KUKA KRL program: EPS_2_251245_SANMH1A_A_20250910012812.src

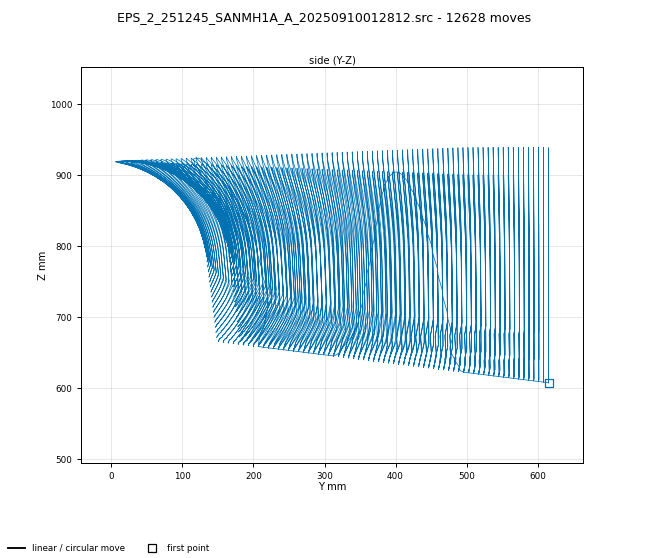
[picture p0: tool path of EPS_2_251245_SANMH1A_A_20250910012812.src, 12628 of 12630 moves have a stored position in this frame; points joined in program order, loops and branches not executed]
&ACCESS RVP
&REL 4
&COMMENT QRS 19112012
&PARAM EDITMASK = *
DEF PART()
EXT BAS (BAS_COMMAND :IN,REAL :IN )
INT I
BAS (#INITMOV,0 )

;KUKA QRS Post kuka4.cps  Date:22-06-2017 !

File_ID=2818

QRS_PRE_INIT()

;Init var - Until changes are made in qrs_pre_init
Outlet_Square_prg=0
Inlet_1_Square_prg=0
Inlet_2_Square_prg=0
Inlet_3_Square_prg=0
Inlet_4_Square_prg=0
Inlet_5_Square_prg=0

Outlet_1={X 0.000, Y 505.360, Z 814.000, B 0.000, E1 0.000 }
Inlet_1={X 0.000, Y 508.180, Z 775.000, B 0.000, E1 175.000 }
Outlet_1_type=251
Inlet_1_type=251
;QRS#1=Sidecore dimensions
;QRS#2=250-10" PVC SDR 35
;QRS#3=250-10" PVC SDR 35
;QRS#4=
;QRS#5=
;QRS#6=
;QRS#7=
;QRS#8=
;QRS#9=14M PSX
;QRS#10=14M PSX
;QRS#11=
;QRS#12=
;QRS#13=
;QRS#14=
;QRS#15=
;QRS#16=1220x127x1219 4'
;QRS#17=EPS Height
;QRS#18=939,5
;QRS#19=*
;QRS#20= UPDATED VERSION 22-06-2017
;QRS#21=*
Outlet_Square=0100
Inlet_1_Square=0100
Inlet_2_Square=0
Inlet_3_Square=0
Inlet_4_Square=0
Inlet_5_Square=0
Mill_Square=1
Outlet_Square_Prg=205
Inlet_1_Square_prg=205

QRS_INIT()

$ADVANCE=5

; T1
PTP {E1 173.423,E2 173.423}
PTP {X 0,Y 615.488,A -85,B 0,C 180,E1 173.423,E2 173.423,E3 0,E4 0,E5 0,E6 0}
QRS_SPEED_INIT()
LIN {X 0,Y 615.488,Z 607.823,A -85,B 0,C 180,E1 173.423,E2 173.423,E3 0,E4 0,E5 0,E6 0} C_VEL
LIN {X 0,Y 615.463,Z 607.814,A -85,B 0,C 180,E1 170.801,E2 170.801} C_VEL
LIN {X 0,Y 615.489,Z 607.808,A -85,B 0,C 180,E1 168.139,E2 168.139} C_VEL
LIN {X 0,Y 615.488,Z 607.825,A -85,B 0,C 180,E1 165.451,E2 165.451} C_VEL
LIN {X 0,Y 615.458,Z 607.816,A -85,B 0,C 180,E1 162.728,E2 162.728} C_VEL
LIN {X 0,Y 615.49,Z 607.808,A -85,B 0,C 180,E1 159.967,E2 159.967} C_VEL
LIN {X 0,Y 615.487,Z 607.825,A -85,B 0,C 180,E1 157.155,E2 157.155} C_VEL
LIN {X 0,Y 615.451,Z 607.816,A -85,B 0,C 180,E1 154.439,E2 154.439} C_VEL
LIN {X 0,Y 615.496,Z 607.811,A -85,B 0,C 180,E1 151.548,E2 151.548} C_VEL
LIN {X 0,Y 615.475,Z 607.824,A -85,B 0,C 180,E1 148.916,E2 148.916} C_VEL
LIN {X 0,Y 615.45,Z 607.819,A -85,B 0,C 180,E1 146.471,E2 146.471} C_VEL
LIN {X 0,Y 615.447,Z 607.816,A -85,B 0,C 180,E1 144.172,E2 144.172} C_VEL
LIN {X 0,Y 615.452,Z 607.814,A -85,B 0,C 180,E1 141.928,E2 141.928} C_VEL
LIN {X 0,Y 615.486,Z 607.812,A -85,B 0,C 180,E1 139.393,E2 139.393} C_VEL
LIN {X 0,Y 615.486,Z 607.824,A -85,B 0,C 180,E1 136.755,E2 136.755} C_VEL
LIN {X 0,Y 615.441,Z 607.819,A -85,B 0,C 180,E1 134.154,E2 134.154} C_VEL
LIN {X 0,Y 615.437,Z 607.819,A -85,B 0,C 180,E1 132.074,E2 132.074} C_VEL
LIN {X 0,Y 615.438,Z 607.817,A -85,B 0,C 180,E1 129.754,E2 129.754} C_VEL
LIN {X 0,Y 615.497,Z 607.816,A -85,B 0,C 180,E1 126.937,E2 126.937} C_VEL
LIN {X 0,Y 615.496,Z 607.823,A -85,B 0,C 180,E1 124.701,E2 124.701} C_VEL
LIN {X 0,Y 615.464,Z 607.823,A -85,B 0,C 180,E1 122.326,E2 122.326} C_VEL
LIN {X 0,Y 615.43,Z 607.82,A -85,B 0,C 180,E1 119.784,E2 119.784} C_VEL
LIN {X 0,Y 615.434,Z 607.822,A -85,B 0,C 180,E1 117.918,E2 117.918} C_VEL
LIN {X 0,Y 615.425,Z 607.82,A -85,B 0,C 180,E1 115.556,E2 115.556} C_VEL
LIN {X 0,Y 615.447,Z 607.824,A -85,B 0,C 180,E1 115.099,E2 115.099} C_VEL
LIN {X 0,Y 615.477,Z 626.453,A -85,B 0,C 180,E1 112.342,E2 112.342} C_VEL
LIN {X 0,Y 615.495,Z 638.775,A -85,B 0,C 180,E1 110.541,E2 110.541} C_VEL
LIN {X 0,Y 615.463,Z 775.158,A -85,B 0,C 180,E1 108.906,E2 108.906} C_VEL
LIN {X 0,Y 615.489,Z 789.394,A -85,B 0,C 180,E1 108.604,E2 108.604} C_VEL
LIN {X 0,Y 615.488,Z 802.541,A -85,B 0,C 180,E1 108.199,E2 108.199} C_VEL
LIN {X 0,Y 615.492,Z 814.87,A -85,B 0,C 180,E1 107.699,E2 107.699} C_VEL
LIN {X 0,Y 615.483,Z 828.082,A -85,B 0,C 180,E1 107.014,E2 107.014} C_VEL
LIN {X 0,Y 615.498,Z 839.221,A -85,B 0,C 180,E1 106.301,E2 106.301} C_VEL
LIN {X 0,Y 615.499,Z 850.82,A -85,B 0,C 180,E1 105.395,E2 105.395} C_VEL
LIN {X 0,Y 615.497,Z 861.349,A -85,B 0,C 180,E1 104.395,E2 104.395} C_VEL
LIN {X 0,Y 615.497,Z 870.257,A -85,B 0,C 180,E1 103.369,E2 103.369} C_VEL
LIN {X 0,Y 615.498,Z 878.577,A -85,B 0,C 180,E1 102.195,E2 102.195} C_VEL
LIN {X 0,Y 615.496,Z 884.373,A -85,B 0,C 180,E1 101.193,E2 101.193} C_VEL
LIN {X 0,Y 615.498,Z 889.088,A -85,B 0,C 180,E1 100.194,E2 100.194} C_VEL
LIN {X 0,Y 615.493,Z 893.953,A -85,B 0,C 180,E1 98.867,E2 98.867} C_VEL
LIN {X 0,Y 615.493,Z 896.596,A -85,B 0,C 180,E1 97.875,E2 97.875} C_VEL
LIN {X 0,Y 615.495,Z 898.88,A -85,B 0,C 180,E1 96.557,E2 96.557} C_VEL
LIN {X 0,Y 615.494,Z 899.826,A -85,B 0,C 180,E1 95.241,E2 95.241} C_VEL
LIN {X 0,Y 615.492,Z 899.459,A -85,B 0,C 180,E1 93.928,E2 93.928} C_VEL
LIN {X 0,Y 615.491,Z 897.783,A -85,B 0,C 180,E1 92.618,E2 92.618} C_VEL
LIN {X 0,Y 615.494,Z 894.753,A -85,B 0,C 180,E1 91.309,E2 91.309} C_VEL
LIN {X 0,Y 615.496,Z 890.297,A -85,B 0,C 180,E1 90,E2 90} C_VEL
LIN {X 0,Y 615.495,Z 885.885,A -85,B 0,C 180,E1 89.019,E2 89.019} C_VEL
LIN {X 0,Y 615.497,Z 880.538,A -85,B 0,C 180,E1 88.037,E2 88.037} C_VEL
LIN {X 0,Y 615.496,Z 872.897,A -85,B 0,C 180,E1 86.891,E2 86.891} C_VEL
LIN {X 0,Y 615.497,Z 863.473,A -85,B 0,C 180,E1 85.744,E2 85.744} C_VEL
LIN {X 0,Y 615.498,Z 853.62,A -85,B 0,C 180,E1 84.759,E2 84.759} C_VEL
LIN {X 0,Y 615.499,Z 842.627,A -85,B 0,C 180,E1 83.855,E2 83.855} C_VEL
LIN {X 0,Y 615.489,Z 830.195,A -85,B 0,C 180,E1 83.022,E2 83.022} C_VEL
LIN {X 0,Y 615.492,Z 818.224,A -85,B 0,C 180,E1 82.372,E2 82.372} C_VEL
LIN {X 0,Y 615.493,Z 804.758,A -85,B 0,C 180,E1 81.794,E2 81.794} C_VEL
LIN {X 0,Y 615.479,Z 790.589,A -85,B 0,C 180,E1 81.339,E2 81.339} C_VEL
LIN {X 0,Y 615.454,Z 776.509,A -85,B 0,C 180,E1 81.028,E2 81.028} C_VEL
LIN {X 0,Y 615.451,Z 738.125,A -85,B 0,C 180,E1 80.552,E2 80.552} C_VEL
LIN {X 0,Y 615.472,Z 638.747,A -85,B 0,C 180,E1 79.364,E2 79.364} C_VEL
LIN {X 0,Y 615.467,Z 620.084,A -85,B 0,C 180,E1 76.63,E2 76.63} C_VEL
LIN {X 0,Y 615.422,Z 607.823,A -85,B 0,C 180,E1 74.793,E2 74.793} C_VEL
LIN {X 0,Y 615.418,Z 607.824,A -85,B 0,C 180,E1 72.727,E2 72.727} C_VEL
LIN {X 0,Y 615.416,Z 607.824,A -85,B 0,C 180,E1 70.66,E2 70.66} C_VEL
LIN {X 0,Y 615.419,Z 607.823,A -85,B 0,C 180,E1 68.565,E2 68.565} C_VEL
LIN {X 0,Y 615.432,Z 607.821,A -85,B 0,C 180,E1 66.005,E2 66.005} C_VEL
LIN {X 0,Y 615.473,Z 607.821,A -85,B 0,C 180,E1 63.555,E2 63.555} C_VEL
LIN {X 0,Y 615.487,Z 607.824,A -85,B 0,C 180,E1 61.342,E2 61.342} C_VEL
LIN {X 0,Y 615.465,Z 607.823,A -85,B 0,C 180,E1 58.918,E2 58.918} C_VEL
LIN {X 0,Y 615.429,Z 607.822,A -85,B 0,C 180,E1 56.475,E2 56.475} C_VEL
LIN {X 0,Y 615.421,Z 607.821,A -85,B 0,C 180,E1 54.176,E2 54.176} C_VEL
LIN {X 0,Y 615.423,Z 607.821,A -85,B 0,C 180,E1 51.927,E2 51.927} C_VEL
LIN {X 0,Y 615.423,Z 607.821,A -85,B 0,C 180,E1 49.919,E2 49.919} C_VEL
LIN {X 0,Y 615.433,Z 607.821,A -85,B 0,C 180,E1 47.642,E2 47.642} C_VEL
LIN {X 0,Y 615.496,Z 607.825,A -85,B 0,C 180,E1 44.932,E2 44.932} C_VEL
LIN {X 0,Y 615.434,Z 607.819,A -85,B 0,C 180,E1 42.074,E2 42.074} C_VEL
LIN {X 0,Y 615.428,Z 607.82,A -85,B 0,C 180,E1 39.755,E2 39.755} C_VEL
LIN {X 0,Y 615.448,Z 607.823,A -85,B 0,C 180,E1 37.245,E2 37.245} C_VEL
LIN {X 0,Y 615.496,Z 607.823,A -85,B 0,C 180,E1 34.701,E2 34.701} C_VEL
LIN {X 0,Y 615.489,Z 607.813,A -85,B 0,C 180,E1 32.331,E2 32.331} C_VEL
LIN {X 0,Y 615.443,Z 607.816,A -85,B 0,C 180,E1 29.787,E2 29.787} C_VEL
LIN {X 0,Y 615.457,Z 607.814,A -85,B 0,C 180,E1 27.917,E2 27.917} C_VEL
LIN {X 0,Y 615.439,Z 607.817,A -85,B 0,C 180,E1 25.559,E2 25.559} C_VEL
LIN {X 0,Y 615.445,Z 607.816,A -85,B 0,C 180,E1 23.558,E2 23.558} C_VEL
LIN {X 0,Y 615.444,Z 607.816,A -85,B 0,C 180,E1 21.434,E2 21.434} C_VEL
LIN {X 0,Y 615.445,Z 607.816,A -85,B 0,C 180,E1 19.34,E2 19.34} C_VEL
LIN {X 0,Y 615.447,Z 607.816,A -85,B 0,C 180,E1 17.272,E2 17.272} C_VEL
LIN {X 0,Y 615.487,Z 607.824,A -85,B 0,C 180,E1 14.549,E2 14.549} C_VEL
LIN {X 0,Y 615.488,Z 607.81,A -85,B 0,C 180,E1 11.861,E2 11.861} C_VEL
LIN {X 0,Y 615.453,Z 607.814,A -85,B 0,C 180,E1 9.2,E2 9.2} C_VEL
LIN {X 0,Y 615.474,Z 607.822,A -85,B 0,C 180,E1 6.557,E2 6.557} C_VEL
LIN {X 0,Y 615.495,Z 607.814,A -85,B 0,C 180,E1 3.929,E2 3.929} C_VEL
LIN {X 0,Y 615.476,Z 607.809,A -85,B 0,C 180,E1 1.309,E2 1.309} C_VEL
LIN {X 0,Y 615.462,Z 607.817,A -85,B 0,C 180,E1 -1.308,E2 -1.308} C_VEL
LIN {X 0,Y 615.492,Z 607.824,A -85,B 0,C 180,E1 -3.928,E2 -3.928} C_VEL
LIN {X 0,Y 615.49,Z 607.808,A -85,B 0,C 180,E1 -6.578,E2 -6.578} C_VEL
LIN {X 0,Y 615.468,Z 607.812,A -85,B 0,C 180,E1 -9.199,E2 -9.199} C_VEL
LIN {X 0,Y 615.486,Z 607.823,A -85,B 0,C 180,E1 -11.861,E2 -11.861} C_VEL
LIN {X 0,Y 615.492,Z 607.81,A -85,B 0,C 180,E1 -14.549,E2 -14.549} C_VEL
LIN {X 0,Y 615.477,Z 607.809,A -85,B 0,C 180,E1 -17.271,E2 -17.271} C_VEL
LIN {X 0,Y 615.491,Z 607.823,A -85,B 0,C 180,E1 -20.033,E2 -20.033} C_VEL
LIN {X 0,Y 615.49,Z 607.808,A -85,B 0,C 180,E1 -22.844,E2 -22.844} C_VEL
LIN {X 0,Y 615.477,Z 607.811,A -85,B 0,C 180,E1 -25.566,E2 -25.566} C_VEL
LIN {X 0,Y 615.496,Z 607.819,A -85,B 0,C 180,E1 -28.451,E2 -28.451} C_VEL
LIN {X 0,Y 615.489,Z 607.807,A -85,B 0,C 180,E1 -31.086,E2 -31.086} C_VEL
LIN {X 0,Y 615.492,Z 607.806,A -85,B 0,C 180,E1 -33.534,E2 -33.534} C_VEL
LIN {X 0,Y 615.49,Z 607.826,A -85,B 0,C 180,E1 -36.425,E2 -36.425} C_VEL
LIN {X 0,Y 615.49,Z 607.809,A -85,B 0,C 180,E1 -39.062,E2 -39.062} C_VEL
LIN {X 0,Y 615.487,Z 607.806,A -85,B 0,C 180,E1 -41.474,E2 -41.474} C_VEL
LIN {X 0,Y 615.484,Z 607.815,A -85,B 0,C 180,E1 -44.15,E2 -44.15} C_VEL
LIN {X 0,Y 615.49,Z 607.814,A -85,B 0,C 180,E1 -46.952,E2 -46.952} C_VEL
LIN {X 0,Y 615.486,Z 607.807,A -85,B 0,C 180,E1 -49.393,E2 -49.393} C_VEL
LIN {X 0,Y 615.487,Z 607.808,A -85,B 0,C 180,E1 -51.988,E2 -51.988} C_VEL
LIN {X 0,Y 615.488,Z 607.816,A -85,B 0,C 180,E1 -54.384,E2 -54.384} C_VEL
LIN {X 0,Y 615.487,Z 607.827,A -85,B 0,C 180,E1 -56.764,E2 -56.764} C_VEL
LIN {X 0,Y 615.484,Z 607.818,A -85,B 0,C 180,E1 -59.08,E2 -59.08} C_VEL
LIN {X 0,Y 615.487,Z 607.808,A -85,B 0,C 180,E1 -61.55,E2 -61.55} C_VEL
LIN {X 0,Y 615.494,Z 607.811,A -85,B 0,C 180,E1 -64.43,E2 -64.43} C_VEL
LIN {X 0,Y 615.488,Z 607.97,A -85,B 0,C 180,E1 -66.162,E2 -66.162} C_VEL
LIN {X 0,Y 615.481,Z 630.471,A -85,B 0,C 180,E1 -68.919,E2 -68.919} C_VEL
LIN {X 0,Y 615.498,Z 653.753,A -85,B 0,C 180,E1 -71.721,E2 -71.721} C_VEL
LIN {X 0,Y 615.495,Z 676.284,A -85,B 0,C 180,E1 -74.392,E2 -74.392} C_VEL
LIN {X 0,Y 615.481,Z 814.24,A -85,B 0,C 180,E1 -76.051,E2 -76.051} C_VEL
LIN {X 0,Y 615.484,Z 827.853,A -85,B 0,C 180,E1 -76.336,E2 -76.336} C_VEL
LIN {X 0,Y 615.491,Z 841.564,A -85,B 0,C 180,E1 -76.757,E2 -76.757} C_VEL
LIN {X 0,Y 615.495,Z 854.834,A -85,B 0,C 180,E1 -77.302,E2 -77.302} C_VEL
LIN {X 0,Y 615.49,Z 867.598,A -85,B 0,C 180,E1 -77.972,E2 -77.972} C_VEL
LIN {X 0,Y 615.499,Z 879.181,A -85,B 0,C 180,E1 -78.724,E2 -78.724} C_VEL
LIN {X 0,Y 615.498,Z 890.747,A -85,B 0,C 180,E1 -79.639,E2 -79.639} C_VEL
LIN {X 0,Y 615.497,Z 901.087,A -85,B 0,C 180,E1 -80.636,E2 -80.636} C_VEL
LIN {X 0,Y 615.497,Z 909.602,A -85,B 0,C 180,E1 -81.629,E2 -81.629} C_VEL
LIN {X 0,Y 615.497,Z 917.726,A -85,B 0,C 180,E1 -82.784,E2 -82.784} C_VEL
LIN {X 0,Y 615.496,Z 923.429,A -85,B 0,C 180,E1 -83.773,E2 -83.773} C_VEL
LIN {X 0,Y 615.495,Z 928.08,A -85,B 0,C 180,E1 -84.759,E2 -84.759} C_VEL
LIN {X 0,Y 615.495,Z 932.901,A -85,B 0,C 180,E1 -86.071,E2 -86.071} C_VEL
LIN {X 0,Y 615.496,Z 936.252,A -85,B 0,C 180,E1 -87.382,E2 -87.382} C_VEL
LIN {X 0,Y 615.489,Z 938.228,A -85,B 0,C 180,E1 -88.691,E2 -88.691} C_VEL
LIN {X 0,Y 615.493,Z 938.889,A -85,B 0,C 180,E1 -90,E2 -90} C_VEL
LIN {X 0,Y 615.489,Z 938.229,A -85,B 0,C 180,E1 -91.309,E2 -91.309} C_VEL
LIN {X 0,Y 615.496,Z 936.252,A -85,B 0,C 180,E1 -92.618,E2 -92.618} C_VEL
LIN {X 0,Y 615.495,Z 932.901,A -85,B 0,C 180,E1 -93.928,E2 -93.928} C_VEL
LIN {X 0,Y 615.495,Z 928.081,A -85,B 0,C 180,E1 -95.241,E2 -95.241} C_VEL
LIN {X 0,Y 615.495,Z 921.628,A -85,B 0,C 180,E1 -96.557,E2 -96.557} C_VEL
LIN {X 0,Y 615.497,Z 914.441,A -85,B 0,C 180,E1 -97.71,E2 -97.71} C_VEL
LIN {X 0,Y 615.497,Z 906.903,A -85,B 0,C 180,E1 -98.702,E2 -98.702} C_VEL
LIN {X 0,Y 615.495,Z 897.853,A -85,B 0,C 180,E1 -99.696,E2 -99.696} C_VEL
LIN {X 0,Y 615.497,Z 887.757,A -85,B 0,C 180,E1 -100.618,E2 -100.618} C_VEL
LIN {X 0,Y 615.498,Z 876.857,A -85,B 0,C 180,E1 -101.443,E2 -101.443} C_VEL
LIN {X 0,Y 615.493,Z 864.705,A -85,B 0,C 180,E1 -102.195,E2 -102.195} C_VEL
LIN {X 0,Y 615.488,Z 851.091,A -85,B 0,C 180,E1 -102.865,E2 -102.865} C_VEL
LIN {X 0,Y 615.489,Z 837.834,A -85,B 0,C 180,E1 -103.369,E2 -103.369} C_VEL
LIN {X 0,Y 615.482,Z 824.286,A -85,B 0,C 180,E1 -103.748,E2 -103.748} C_VEL
LIN {X 0,Y 615.482,Z 810.17,A -85,B 0,C 180,E1 -104.007,E2 -104.007} C_VEL
LIN {X 0,Y 615.495,Z 676.286,A -85,B 0,C 180,E1 -105.608,E2 -105.608} C_VEL
LIN {X 0,Y 615.489,Z 652.401,A -85,B 0,C 180,E1 -108.441,E2 -108.441} C_VEL
LIN {X 0,Y 615.482,Z 629.028,A -85,B 0,C 180,E1 -111.256,E2 -111.256} C_VEL
LIN {X 0,Y 615.487,Z 607.807,A -85,B 0,C 180,E1 -113.866,E2 -113.866} C_VEL
LIN {X 0,Y 615.486,Z 607.808,A -85,B 0,C 180,E1 -116.444,E2 -116.444} C_VEL
LIN {X 0,Y 615.485,Z 607.811,A -85,B 0,C 180,E1 -118.658,E2 -118.658} C_VEL
LIN {X 0,Y 615.488,Z 607.822,A -85,B 0,C 180,E1 -121.086,E2 -121.086} C_VEL
LIN {X 0,Y 615.492,Z 607.807,A -85,B 0,C 180,E1 -124.022,E2 -124.022} C_VEL
LIN {X 0,Y 615.484,Z 607.807,A -85,B 0,C 180,E1 -126.425,E2 -126.425} C_VEL
LIN {X 0,Y 615.481,Z 607.818,A -85,B 0,C 180,E1 -129.061,E2 -129.061} C_VEL
LIN {X 0,Y 615.497,Z 607.824,A -85,B 0,C 180,E1 -131.473,E2 -131.473} C_VEL
LIN {X 0,Y 615.495,Z 607.807,A -85,B 0,C 180,E1 -134.149,E2 -134.149} C_VEL
LIN {X 0,Y 615.492,Z 607.809,A -85,B 0,C 180,E1 -136.952,E2 -136.952} C_VEL
LIN {X 0,Y 615.489,Z 607.82,A -85,B 0,C 180,E1 -139.394,E2 -139.394} C_VEL
LIN {X 0,Y 615.484,Z 607.816,A -85,B 0,C 180,E1 -141.989,E2 -141.989} C_VEL
LIN {X 0,Y 615.491,Z 607.807,A -85,B 0,C 180,E1 -144.384,E2 -144.384} C_VEL
LIN {X 0,Y 615.491,Z 607.805,A -85,B 0,C 180,E1 -146.764,E2 -146.764} C_VEL
LIN {X 0,Y 615.49,Z 607.808,A -85,B 0,C 180,E1 -149.08,E2 -149.08} C_VEL
LIN {X 0,Y 615.494,Z 607.817,A -85,B 0,C 180,E1 -151.549,E2 -151.549} C_VEL
LIN {X 0,Y 615.48,Z 607.812,A -85,B 0,C 180,E1 -154.433,E2 -154.433} C_VEL
LIN {X 0,Y 615.49,Z 607.807,A -85,B 0,C 180,E1 -157.156,E2 -157.156} C_VEL
LIN {X 0,Y 615.49,Z 607.827,A -85,B 0,C 180,E1 -159.967,E2 -159.967} C_VEL
LIN {X 0,Y 615.48,Z 607.81,A -85,B 0,C 180,E1 -162.729,E2 -162.729} C_VEL
LIN {X 0,Y 615.492,Z 607.808,A -85,B 0,C 180,E1 -165.451,E2 -165.451} C_VEL
LIN {X 0,Y 615.489,Z 607.827,A -85,B 0,C 180,E1 -168.139,E2 -168.139} C_VEL
LIN {X 0,Y 615.473,Z 607.812,A -85,B 0,C 180,E1 -170.801,E2 -170.801} C_VEL
LIN {X 0,Y 615.491,Z 607.806,A -85,B 0,C 180,E1 -173.444,E2 -173.444} C_VEL
LIN {X 0,Y 615.495,Z 607.819,A -85,B 0,C 180,E1 -176.072,E2 -176.072} C_VEL
LIN {X 0,Y 615.472,Z 607.818,A -85,B 0,C 180,E1 -178.692,E2 -178.692} C_VEL
LIN {X 0,Y 615.479,Z 607.808,A -85,B 0,C 180,E1 -181.309,E2 -181.309} C_VEL
LIN {X 0,Y 615.495,Z 607.81,A -85,B 0,C 180,E1 -183.929,E2 -183.929} C_VEL
LIN {X 0,Y 615.488,Z 607.823,A -85,B 0,C 180,E1 -186.577,E2 -186.577} C_VEL
LIN {X 0,Y 614.795,Z 607.961,A -85,B 0,C 180,E1 -187.123,E2 -187.123} C_VEL
LIN {X 0,Y 611.945,Z 608.38,A -85,B 0,C 180,E1 -188.009,E2 -188.009} C_VEL
LIN {X 0,Y 609.556,Z 608.688,A -85,B 0,C 180,E1 -188.722,E2 -188.722} C_VEL
LIN {X 0,Y 608.532,Z 608.803,A -85,B 0,C 180,E1 -189.271,E2 -189.271} C_VEL
LIN {X 0,Y 608.449,Z 608.812,A -85,B 0,C 180,E1 -189.457,E2 -189.457} C_VEL
LIN {X 0,Y 608.466,Z 608.812,A -85,B 0,C 180,E1 -192,E2 -192} C_VEL
LIN {X 0,Y 608.47,Z 608.819,A -85,B 0,C 180,E1 -194.721,E2 -194.721} C_VEL
LIN {X 0,Y 608.437,Z 608.814,A -85,B 0,C 180,E1 -197.477,E2 -197.477} C_VEL
LIN {X 0,Y 608.436,Z 608.814,A -85,B 0,C 180,E1 -199.571,E2 -199.571} C_VEL
LIN {X 0,Y 608.48,Z 608.813,A -85,B 0,C 180,E1 -202.405,E2 -202.405} C_VEL
LIN {X 0,Y 608.455,Z 608.818,A -85,B 0,C 180,E1 -204.571,E2 -204.571} C_VEL
LIN {X 0,Y 608.433,Z 608.815,A -85,B 0,C 180,E1 -207.519,E2 -207.519} C_VEL
LIN {X 0,Y 608.445,Z 608.812,A -85,B 0,C 180,E1 -209.968,E2 -209.968} C_VEL
LIN {X 0,Y 608.454,Z 608.822,A -85,B 0,C 180,E1 -212.88,E2 -212.88} C_VEL
LIN {X 0,Y 608.426,Z 608.821,A -85,B 0,C 180,E1 -215.279,E2 -215.279} C_VEL
LIN {X 0,Y 608.443,Z 608.814,A -85,B 0,C 180,E1 -217.749,E2 -217.749} C_VEL
LIN {X 0,Y 608.435,Z 608.814,A -85,B 0,C 180,E1 -220.327,E2 -220.327} C_VEL
LIN {X 0,Y 608.472,Z 608.817,A -85,B 0,C 180,E1 -223.309,E2 -223.309} C_VEL
LIN {X 0,Y 608.435,Z 608.814,A -85,B 0,C 180,E1 -226.127,E2 -226.127} C_VEL
LIN {X 0,Y 608.452,Z 608.816,A -85,B 0,C 180,E1 -228.823,E2 -228.823} C_VEL
LIN {X 0,Y 608.436,Z 608.817,A -85,B 0,C 180,E1 -231.764,E2 -231.764} C_VEL
LIN {X 0,Y 608.431,Z 608.816,A -85,B 0,C 180,E1 -233.957,E2 -233.957} C_VEL
LIN {X 0,Y 608.413,Z 608.816,A -85,B 0,C 180,E1 -236.326,E2 -236.326} C_VEL
LIN {X 0,Y 608.439,Z 608.814,A -85,B 0,C 180,E1 -238.734,E2 -238.734} C_VEL
LIN {X 0,Y 608.434,Z 608.821,A -85,B 0,C 180,E1 -241.732,E2 -241.732} C_VEL
LIN {X 0,Y 608.424,Z 608.817,A -85,B 0,C 180,E1 -244.289,E2 -244.289} C_VEL
LIN {X 0,Y 608.453,Z 609.014,A -85,B 0,C 180,E1 -244.836,E2 -244.836} C_VEL
LIN {X 0,Y 608.511,Z 625.068,A -85,B 0,C 180,E1 -247.238,E2 -247.238} C_VEL
LIN {X 0,Y 608.498,Z 638.922,A -85,B 0,C 180,E1 -249.283,E2 -249.283} C_VEL
LIN {X 0,Y 608.588,Z 756.65,A -85,B 0,C 180,E1 -250.697,E2 -250.697} C_VEL
LIN {X 0,Y 608.588,Z 777.773,A -85,B 0,C 180,E1 -250.982,E2 -250.982} C_VEL
LIN {X 0,Y 608.58,Z 792.407,A -85,B 0,C 180,E1 -251.323,E2 -251.323} C_VEL
LIN {X 0,Y 608.575,Z 806.351,A -85,B 0,C 180,E1 -251.791,E2 -251.791} C_VEL
LIN {X 0,Y 608.543,Z 819.031,A -85,B 0,C 180,E1 -252.353,E2 -252.353} C_VEL
LIN {X 0,Y 608.527,Z 831.481,A -85,B 0,C 180,E1 -253.045,E2 -253.045} C_VEL
LIN {X 0,Y 608.509,Z 842.188,A -85,B 0,C 180,E1 -253.774,E2 -253.774} C_VEL
LIN {X 0,Y 608.491,Z 852.284,A -85,B 0,C 180,E1 -254.595,E2 -254.595} C_VEL
LIN {X 0,Y 608.475,Z 862.8,A -85,B 0,C 180,E1 -255.621,E2 -255.621} C_VEL
LIN {X 0,Y 608.462,Z 871.428,A -85,B 0,C 180,E1 -256.644,E2 -256.644} C_VEL
LIN {X 0,Y 608.441,Z 879.631,A -85,B 0,C 180,E1 -257.831,E2 -257.831} C_VEL
LIN {X 0,Y 608.432,Z 886.464,A -85,B 0,C 180,E1 -259.065,E2 -259.065} C_VEL
LIN {X 0,Y 608.428,Z 892.015,A -85,B 0,C 180,E1 -260.358,E2 -260.358} C_VEL
LIN {X 0,Y 608.426,Z 895.325,A -85,B 0,C 180,E1 -261.364,E2 -261.364} C_VEL
LIN {X 0,Y 608.421,Z 898.403,A -85,B 0,C 180,E1 -262.7,E2 -262.7} C_VEL
LIN {X 0,Y 608.432,Z 900.085,A -85,B 0,C 180,E1 -264.033,E2 -264.033} C_VEL
LIN {X 0,Y 608.424,Z 900.432,A -85,B 0,C 180,E1 -265.362,E2 -265.362} C_VEL
LIN {X 0,Y 608.416,Z 899.453,A -85,B 0,C 180,E1 -266.689,E2 -266.689} C_VEL
LIN {X 0,Y 608.443,Z 897.137,A -85,B 0,C 180,E1 -268.014,E2 -268.014} C_VEL
LIN {X 0,Y 608.437,Z 893.423,A -85,B 0,C 180,E1 -269.338,E2 -269.338} C_VEL
LIN {X 0,Y 608.437,Z 888.216,A -85,B 0,C 180,E1 -270.662,E2 -270.662} C_VEL
LIN {X 0,Y 608.441,Z 883.177,A -85,B 0,C 180,E1 -271.655,E2 -271.655} C_VEL
LIN {X 0,Y 608.446,Z 876.008,A -85,B 0,C 180,E1 -272.814,E2 -272.814} C_VEL
LIN {X 0,Y 608.455,Z 867.176,A -85,B 0,C 180,E1 -273.974,E2 -273.974} C_VEL
LIN {X 0,Y 608.474,Z 857.942,A -85,B 0,C 180,E1 -274.97,E2 -274.97} C_VEL
LIN {X 0,Y 608.497,Z 846.693,A -85,B 0,C 180,E1 -275.967,E2 -275.967} C_VEL
LIN {X 0,Y 608.535,Z 834.522,A -85,B 0,C 180,E1 -276.849,E2 -276.849} C_VEL
LIN {X 0,Y 608.541,Z 822.682,A -85,B 0,C 180,E1 -277.549,E2 -277.549} C_VEL
LIN {X 0,Y 608.572,Z 810.417,A -85,B 0,C 180,E1 -278.133,E2 -278.133} C_VEL
LIN {X 0,Y 608.585,Z 796.855,A -85,B 0,C 180,E1 -278.634,E2 -278.634} C_VEL
LIN {X 0,Y 608.566,Z 782.762,A -85,B 0,C 180,E1 -279.011,E2 -279.011} C_VEL
LIN {X 0,Y 608.57,Z 769.26,A -85,B 0,C 180,E1 -279.242,E2 -279.242} C_VEL
LIN {X 0,Y 608.587,Z 639.744,A -85,B 0,C 180,E1 -280.792,E2 -280.792} C_VEL
LIN {X 0,Y 608.477,Z 638.817,A -85,B 0,C 180,E1 -280.823,E2 -280.823} C_VEL
LIN {X 0,Y 608.487,Z 621.681,A -85,B 0,C 180,E1 -283.356,E2 -283.356} C_VEL
LIN {X 0,Y 608.423,Z 608.855,A -85,B 0,C 180,E1 -285.279,E2 -285.279} C_VEL
LIN {X 0,Y 608.398,Z 608.819,A -85,B 0,C 180,E1 -287.478,E2 -287.478} C_VEL
LIN {X 0,Y 608.397,Z 608.819,A -85,B 0,C 180,E1 -289.573,E2 -289.573} C_VEL
LIN {X 0,Y 608.418,Z 608.816,A -85,B 0,C 180,E1 -291.694,E2 -291.694} C_VEL
LIN {X 0,Y 608.431,Z 608.823,A -85,B 0,C 180,E1 -294.572,E2 -294.572} C_VEL
LIN {X 0,Y 608.405,Z 608.818,A -85,B 0,C 180,E1 -297.52,E2 -297.52} C_VEL
LIN {X 0,Y 608.407,Z 608.817,A -85,B 0,C 180,E1 -299.783,E2 -299.783} C_VEL
LIN {X 0,Y 608.441,Z 608.819,A -85,B 0,C 180,E1 -302.518,E2 -302.518} C_VEL
LIN {X 0,Y 608.417,Z 608.82,A -85,B 0,C 180,E1 -305.28,E2 -305.28} C_VEL
LIN {X 0,Y 608.404,Z 608.818,A -85,B 0,C 180,E1 -307.751,E2 -307.751} C_VEL
LIN {X 0,Y 608.405,Z 608.819,A -85,B 0,C 180,E1 -310.323,E2 -310.323} C_VEL
LIN {X 0,Y 608.453,Z 608.822,A -85,B 0,C 180,E1 -312.96,E2 -312.96} C_VEL
LIN {X 0,Y 608.415,Z 608.817,A -85,B 0,C 180,E1 -315.74,E2 -315.74} C_VEL
LIN {X 0,Y 608.418,Z 608.816,A -85,B 0,C 180,E1 -317.935,E2 -317.935} C_VEL
LIN {X 0,Y 608.424,Z 608.819,A -85,B 0,C 180,E1 -320.708,E2 -320.708} C_VEL
LIN {X 0,Y 608.445,Z 608.822,A -85,B 0,C 180,E1 -323.084,E2 -323.084} C_VEL
LIN {X 0,Y 608.466,Z 608.816,A -85,B 0,C 180,E1 -325.53,E2 -325.53} C_VEL
LIN {X 0,Y 608.453,Z 608.813,A -85,B 0,C 180,E1 -327.904,E2 -327.904} C_VEL
LIN {X 0,Y 608.431,Z 608.814,A -85,B 0,C 180,E1 -330.218,E2 -330.218} C_VEL
LIN {X 0,Y 608.422,Z 608.816,A -85,B 0,C 180,E1 -332.48,E2 -332.48} C_VEL
LIN {X 0,Y 608.447,Z 608.823,A -85,B 0,C 180,E1 -335.428,E2 -335.428} C_VEL
LIN {X 0,Y 608.449,Z 608.812,A -85,B 0,C 180,E1 -338.307,E2 -338.307} C_VEL
LIN {X 0,Y 608.428,Z 608.815,A -85,B 0,C 180,E1 -340.428,E2 -340.428} C_VEL
LIN {X 0,Y 608.43,Z 608.814,A -85,B 0,C 180,E1 -342.522,E2 -342.522} C_VEL
LIN {X 0,Y 608.468,Z 608.816,A -85,B 0,C 180,E1 -345.279,E2 -345.279} C_VEL
LIN {X 0,Y 608.463,Z 608.814,A -85,B 0,C 180,E1 -348,E2 -348} C_VEL
LIN {X 0,Y 608.447,Z 608.812,A -85,B 0,C 180,E1 -350.694,E2 -350.694} C_VEL
LIN {X 0,Y 608.433,Z 608.814,A -85,B 0,C 180,E1 -352.7,E2 -352.7} C_VEL
LIN {X 0,Y 608.437,Z 608.818,A -85,B 0,C 180,E1 -355.362,E2 -355.362} C_VEL
LIN {X 0,Y 608.466,Z 608.817,A -85,B 0,C 180,E1 -358.014,E2 -358.014} C_VEL
LIN {X 0,Y 608.476,Z 608.809,A -85,B 0,C 180,E1 -360.662,E2 -360.662} C_VEL
LIN {X 0,Y 608.458,Z 608.813,A -85,B 0,C 180,E1 -363.311,E2 -363.311} C_VEL
LIN {X 0,Y 608.472,Z 608.819,A -85,B 0,C 180,E1 -365.967,E2 -365.967} C_VEL
LIN {X 0,Y 608.46,Z 608.812,A -85,B 0,C 180,E1 -368.636,E2 -368.636} C_VEL
LIN {X 0,Y 608.437,Z 608.815,A -85,B 0,C 180,E1 -371.324,E2 -371.324} C_VEL
LIN {X 0,Y 608.473,Z 608.821,A -85,B 0,C 180,E1 -374.037,E2 -374.037} C_VEL
LIN {X 0,Y 608.476,Z 608.81,A -85,B 0,C 180,E1 -376.783,E2 -376.783} C_VEL
LIN {X 0,Y 608.449,Z 608.814,A -85,B 0,C 180,E1 -379.571,E2 -379.571} C_VEL
LIN {X 0,Y 608.48,Z 608.815,A -85,B 0,C 180,E1 -382.405,E2 -382.405} C_VEL
LIN {X 0,Y 608.459,Z 608.816,A -85,B 0,C 180,E1 -384.571,E2 -384.571} C_VEL
LIN {X 0,Y 608.482,Z 608.808,A -85,B 0,C 180,E1 -387.207,E2 -387.207} C_VEL
LIN {X 0,Y 608.462,Z 608.816,A -85,B 0,C 180,E1 -389.97,E2 -389.97} C_VEL
LIN {X 0,Y 608.463,Z 608.813,A -85,B 0,C 180,E1 -392.879,E2 -392.879} C_VEL
LIN {X 0,Y 608.451,Z 608.812,A -85,B 0,C 180,E1 -395.277,E2 -395.277} C_VEL
LIN {X 0,Y 608.468,Z 608.811,A -85,B 0,C 180,E1 -397.746,E2 -397.746} C_VEL
LIN {X 0,Y 608.452,Z 608.82,A -85,B 0,C 180,E1 -400.329,E2 -400.329} C_VEL
LIN {X 0,Y 608.474,Z 608.809,A -85,B 0,C 180,E1 -403.309,E2 -403.309} C_VEL
LIN {X 0,Y 608.472,Z 608.813,A -85,B 0,C 180,E1 -406.131,E2 -406.131} C_VEL
LIN {X 0,Y 608.463,Z 608.818,A -85,B 0,C 180,E1 -408.824,E2 -408.824} C_VEL
LIN {X 0,Y 608.47,Z 608.81,A -85,B 0,C 180,E1 -411.759,E2 -411.759} C_VEL
LIN {X 0,Y 608.48,Z 608.809,A -85,B 0,C 180,E1 -413.95,E2 -413.95} C_VEL
LIN {X 0,Y 608.467,Z 608.814,A -85,B 0,C 180,E1 -416.329,E2 -416.329} C_VEL
LIN {X 0,Y 608.48,Z 608.819,A -85,B 0,C 180,E1 -418.727,E2 -418.727} C_VEL
LIN {X 0,Y 608.473,Z 608.811,A -85,B 0,C 180,E1 -421.38,E2 -421.38} C_VEL
LIN {X 0,Y 608.481,Z 608.81,A -85,B 0,C 180,E1 -424.277,E2 -424.277} C_VEL
LIN {X 0,Y 608.475,Z 608.889,A -85,B 0,C 180,E1 -425.985,E2 -425.985} C_VEL
LIN {X 0,Y 608.599,Z 621.803,A -85,B 0,C 180,E1 -427.599,E2 -427.599} C_VEL
LIN {X 0,Y 608.576,Z 644.918,A -85,B 0,C 180,E1 -430.433,E2 -430.433} C_VEL
LIN {X 0,Y 608.521,Z 668.034,A -85,B 0,C 180,E1 -433.218,E2 -433.218} C_VEL
LIN {X 0,Y 608.537,Z 676.431,A -85,B 0,C 180,E1 -434.22,E2 -434.22} C_VEL
LIN {X 0,Y 608.601,Z 814.446,A -85,B 0,C 180,E1 -435.894,E2 -435.894} C_VEL
LIN {X 0,Y 608.581,Z 828.62,A -85,B 0,C 180,E1 -436.199,E2 -436.199} C_VEL
LIN {X 0,Y 608.578,Z 842.707,A -85,B 0,C 180,E1 -436.646,E2 -436.646} C_VEL
LIN {X 0,Y 608.556,Z 854.88,A -85,B 0,C 180,E1 -437.155,E2 -437.155} C_VEL
LIN {X 0,Y 608.519,Z 867.678,A -85,B 0,C 180,E1 -437.832,E2 -437.832} C_VEL
LIN {X 0,Y 608.499,Z 880.469,A -85,B 0,C 180,E1 -438.677,E2 -438.677} C_VEL
LIN {X 0,Y 608.496,Z 890.929,A -85,B 0,C 180,E1 -439.519,E2 -439.519} C_VEL
LIN {X 0,Y 608.479,Z 901.333,A -85,B 0,C 180,E1 -440.527,E2 -440.527} C_VEL
LIN {X 0,Y 608.464,Z 909.913,A -85,B 0,C 180,E1 -441.531,E2 -441.531} C_VEL
LIN {X 0,Y 608.461,Z 918.113,A -85,B 0,C 180,E1 -442.7,E2 -442.7} C_VEL
LIN {X 0,Y 608.443,Z 924.545,A -85,B 0,C 180,E1 -443.831,E2 -443.831} C_VEL
LIN {X 0,Y 608.435,Z 929.961,A -85,B 0,C 180,E1 -445.03,E2 -445.03} C_VEL
LIN {X 0,Y 608.433,Z 933.441,A -85,B 0,C 180,E1 -446.026,E2 -446.026} C_VEL
LIN {X 0,Y 608.424,Z 936.831,A -85,B 0,C 180,E1 -447.352,E2 -447.352} C_VEL
LIN {X 0,Y 608.442,Z 938.83,A -85,B 0,C 180,E1 -448.676,E2 -448.676} C_VEL
LIN {X 0,Y 608.433,Z 939.5,A -85,B 0,C 180,E1 -450,E2 -450} C_VEL
LIN {X 0,Y 608.442,Z 938.83,A -85,B 0,C 180,E1 -451.324,E2 -451.324} C_VEL
LIN {X 0,Y 608.424,Z 936.831,A -85,B 0,C 180,E1 -452.648,E2 -452.648} C_VEL
LIN {X 0,Y 608.433,Z 933.441,A -85,B 0,C 180,E1 -453.974,E2 -453.974} C_VEL
LIN {X 0,Y 608.439,Z 928.568,A -85,B 0,C 180,E1 -455.302,E2 -455.302} C_VEL
LIN {X 0,Y 608.445,Z 922.211,A -85,B 0,C 180,E1 -456.603,E2 -456.603} C_VEL
LIN {X 0,Y 608.453,Z 914.798,A -85,B 0,C 180,E1 -457.8,E2 -457.8} C_VEL
LIN {X 0,Y 608.473,Z 905.823,A -85,B 0,C 180,E1 -458.971,E2 -458.971} C_VEL
LIN {X 0,Y 608.472,Z 896.391,A -85,B 0,C 180,E1 -459.977,E2 -459.977} C_VEL
LIN {X 0,Y 608.506,Z 885.047,A -85,B 0,C 180,E1 -460.973,E2 -460.973} C_VEL
LIN {X 0,Y 608.531,Z 873.147,A -85,B 0,C 180,E1 -461.829,E2 -461.829} C_VEL
LIN {X 0,Y 608.535,Z 860.072,A -85,B 0,C 180,E1 -462.591,E2 -462.591} C_VEL
LIN {X 0,Y 608.557,Z 847.172,A -85,B 0,C 180,E1 -463.184,E2 -463.184} C_VEL
LIN {X 0,Y 608.584,Z 833.18,A -85,B 0,C 180,E1 -463.673,E2 -463.673} C_VEL
LIN {X 0,Y 608.598,Z 819.451,A -85,B 0,C 180,E1 -464.013,E2 -464.013} C_VEL
LIN {X 0,Y 608.622,Z 803.162,A -85,B 0,C 180,E1 -464.257,E2 -464.257} C_VEL
LIN {X 0,Y 608.529,Z 676.432,A -85,B 0,C 180,E1 -465.78,E2 -465.78} C_VEL
LIN {X 0,Y 608.551,Z 653.767,A -85,B 0,C 180,E1 -468.496,E2 -468.496} C_VEL
LIN {X 0,Y 608.573,Z 630.473,A -85,B 0,C 180,E1 -471.332,E2 -471.332} C_VEL
LIN {X 0,Y 608.642,Z 610.247,A -85,B 0,C 180,E1 -473.838,E2 -473.838} C_VEL
LIN {X 0,Y 608.477,Z 608.811,A -85,B 0,C 180,E1 -474.043,E2 -474.043} C_VEL
LIN {X 0,Y 608.449,Z 608.817,A -85,B 0,C 180,E1 -476.774,E2 -476.774} C_VEL
LIN {X 0,Y 608.472,Z 608.817,A -85,B 0,C 180,E1 -479.02,E2 -479.02} C_VEL
LIN {X 0,Y 608.479,Z 608.819,A -85,B 0,C 180,E1 -481.316,E2 -481.316} C_VEL
LIN {X 0,Y 608.477,Z 608.812,A -85,B 0,C 180,E1 -483.735,E2 -483.735} C_VEL
LIN {X 0,Y 608.479,Z 608.809,A -85,B 0,C 180,E1 -486.09,E2 -486.09} C_VEL
LIN {X 0,Y 608.472,Z 608.81,A -85,B 0,C 180,E1 -488.588,E2 -488.588} C_VEL
LIN {X 0,Y 608.47,Z 608.819,A -85,B 0,C 180,E1 -491.343,E2 -491.343} C_VEL
LIN {X 0,Y 608.464,Z 608.811,A -85,B 0,C 180,E1 -494.265,E2 -494.265} C_VEL
LIN {X 0,Y 608.459,Z 608.814,A -85,B 0,C 180,E1 -497.041,E2 -497.041} C_VEL
LIN {X 0,Y 608.453,Z 608.821,A -85,B 0,C 180,E1 -499.697,E2 -499.697} C_VEL
LIN {X 0,Y 608.469,Z 608.811,A -85,B 0,C 180,E1 -502.254,E2 -502.254} C_VEL
LIN {X 0,Y 608.487,Z 608.809,A -85,B 0,C 180,E1 -505.09,E2 -505.09} C_VEL
LIN {X 0,Y 608.473,Z 608.817,A -85,B 0,C 180,E1 -507.906,E2 -507.906} C_VEL
LIN {X 0,Y 608.466,Z 608.814,A -85,B 0,C 180,E1 -510.22,E2 -510.22} C_VEL
LIN {X 0,Y 608.482,Z 608.808,A -85,B 0,C 180,E1 -512.792,E2 -512.792} C_VEL
LIN {X 0,Y 608.485,Z 608.819,A -85,B 0,C 180,E1 -515.846,E2 -515.846} C_VEL
LIN {X 0,Y 608.469,Z 608.814,A -85,B 0,C 180,E1 -518.309,E2 -518.309} C_VEL
LIN {X 0,Y 608.458,Z 608.811,A -85,B 0,C 180,E1 -521.131,E2 -521.131} C_VEL
LIN {X 0,Y 608.466,Z 608.819,A -85,B 0,C 180,E1 -523.906,E2 -523.906} C_VEL
LIN {X 0,Y 608.458,Z 608.813,A -85,B 0,C 180,E1 -526.644,E2 -526.644} C_VEL
LIN {X 0,Y 608.467,Z 608.81,A -85,B 0,C 180,E1 -529.35,E2 -529.35} C_VEL
LIN {X 0,Y 608.478,Z 608.817,A -85,B 0,C 180,E1 -532.033,E2 -532.033} C_VEL
LIN {X 0,Y 608.452,Z 608.815,A -85,B 0,C 180,E1 -534.698,E2 -534.698} C_VEL
LIN {X 0,Y 608.483,Z 608.808,A -85,B 0,C 180,E1 -537.352,E2 -537.352} C_VEL
LIN {X 0,Y 608.478,Z 608.814,A -85,B 0,C 180,E1 -540,E2 -540} C_VEL
LIN {X 0,Y 608.47,Z 608.816,A -85,B 0,C 180,E1 -542.648,E2 -542.648} C_VEL
LIN {X 0,Y 608.451,Z 608.812,A -85,B 0,C 180,E1 -545.302,E2 -545.302} C_VEL
LIN {X 0,Y 608.485,Z 608.81,A -85,B 0,C 180,E1 -547.967,E2 -547.967} C_VEL
LIN {X 0,Y 608.449,Z 608.812,A -85,B 0,C 180,E1 -549.457,E2 -549.457} C_VEL
LIN {X 0,Y 607.785,Z 608.899,A -85,B 0,C 180,E1 -550.01,E2 -550.01} C_VEL
LIN {X 0,Y 604.939,Z 609.254,A -85,B 0,C 180,E1 -550.907,E2 -550.907} C_VEL
LIN {X 0,Y 602.532,Z 609.553,A -85,B 0,C 180,E1 -551.628,E2 -551.628} C_VEL
LIN {X 0,Y 601.496,Z 609.683,A -85,B 0,C 180,E1 -552.185,E2 -552.185} C_VEL
LIN {X 0,Y 601.41,Z 609.692,A -85,B 0,C 180,E1 -552.373,E2 -552.373} C_VEL
LIN {X 0,Y 601.423,Z 609.693,A -85,B 0,C 180,E1 -554.897,E2 -554.897} C_VEL
LIN {X 0,Y 601.429,Z 609.692,A -85,B 0,C 180,E1 -556.986,E2 -556.986} C_VEL
LIN {X 0,Y 601.399,Z 609.69,A -85,B 0,C 180,E1 -559.81,E2 -559.81} C_VEL
LIN {X 0,Y 601.418,Z 609.696,A -85,B 0,C 180,E1 -562.606,E2 -562.606} C_VEL
LIN {X 0,Y 601.394,Z 609.701,A -85,B 0,C 180,E1 -564.879,E2 -564.879} C_VEL
LIN {X 0,Y 601.391,Z 609.694,A -85,B 0,C 180,E1 -567.358,E2 -567.358} C_VEL
LIN {X 0,Y 601.401,Z 609.692,A -85,B 0,C 180,E1 -569.394,E2 -569.394} C_VEL
LIN {X 0,Y 601.396,Z 609.691,A -85,B 0,C 180,E1 -571.728,E2 -571.728} C_VEL
LIN {X 0,Y 601.413,Z 609.689,A -85,B 0,C 180,E1 -574.12,E2 -574.12} C_VEL
LIN {X 0,Y 601.435,Z 609.691,A -85,B 0,C 180,E1 -577.382,E2 -577.382} C_VEL
LIN {X 0,Y 601.4,Z 609.69,A -85,B 0,C 180,E1 -579.996,E2 -579.996} C_VEL
LIN {X 0,Y 601.39,Z 609.695,A -85,B 0,C 180,E1 -582.673,E2 -582.673} C_VEL
LIN {X 0,Y 601.402,Z 609.696,A -85,B 0,C 180,E1 -585.48,E2 -585.48} C_VEL
LIN {X 0,Y 601.409,Z 609.69,A -85,B 0,C 180,E1 -588.409,E2 -588.409} C_VEL
LIN {X 0,Y 601.402,Z 609.697,A -85,B 0,C 180,E1 -591.533,E2 -591.533} C_VEL
LIN {X 0,Y 601.392,Z 609.695,A -85,B 0,C 180,E1 -593.741,E2 -593.741} C_VEL
LIN {X 0,Y 601.406,Z 609.691,A -85,B 0,C 180,E1 -596.069,E2 -596.069} C_VEL
LIN {X 0,Y 601.39,Z 609.692,A -85,B 0,C 180,E1 -598.551,E2 -598.551} C_VEL
LIN {X 0,Y 601.434,Z 609.696,A -85,B 0,C 180,E1 -601.373,E2 -601.373} C_VEL
LIN {X 0,Y 601.375,Z 609.695,A -85,B 0,C 180,E1 -604.38,E2 -604.38} C_VEL
LIN {X 0,Y 601.387,Z 609.778,A -85,B 0,C 180,E1 -604.705,E2 -604.705} C_VEL
LIN {X 0,Y 601.509,Z 619.788,A -85,B 0,C 180,E1 -606.228,E2 -606.228} C_VEL
LIN {X 0,Y 601.509,Z 638.445,A -85,B 0,C 180,E1 -609.024,E2 -609.024} C_VEL
LIN {X 0,Y 601.495,Z 638.915,A -85,B 0,C 180,E1 -609.094,E2 -609.094} C_VEL
LIN {X 0,Y 601.838,Z 644.286,A -85,B 0,C 180,E1 -609.172,E2 -609.172} C_VEL
LIN {X 0,Y 601.719,Z 775.68,A -85,B 0,C 180,E1 -610.778,E2 -610.778} C_VEL
LIN {X 0,Y 601.704,Z 789.973,A -85,B 0,C 180,E1 -611.094,E2 -611.094} C_VEL
LIN {X 0,Y 601.652,Z 802.874,A -85,B 0,C 180,E1 -611.502,E2 -611.502} C_VEL
LIN {X 0,Y 601.591,Z 815.987,A -85,B 0,C 180,E1 -612.054,E2 -612.054} C_VEL
LIN {X 0,Y 601.551,Z 829.026,A -85,B 0,C 180,E1 -612.755,E2 -612.755} C_VEL
LIN {X 0,Y 601.5,Z 841.505,A -85,B 0,C 180,E1 -613.591,E2 -613.591} C_VEL
LIN {X 0,Y 601.485,Z 851.592,A -85,B 0,C 180,E1 -614.411,E2 -614.411} C_VEL
LIN {X 0,Y 601.443,Z 862.236,A -85,B 0,C 180,E1 -615.45,E2 -615.45} C_VEL
LIN {X 0,Y 601.4,Z 870.973,A -85,B 0,C 180,E1 -616.484,E2 -616.484} C_VEL
LIN {X 0,Y 601.381,Z 879.272,A -85,B 0,C 180,E1 -617.686,E2 -617.686} C_VEL
LIN {X 0,Y 601.362,Z 885.902,A -85,B 0,C 180,E1 -618.877,E2 -618.877} C_VEL
LIN {X 0,Y 601.345,Z 890.512,A -85,B 0,C 180,E1 -619.904,E2 -619.904} C_VEL
LIN {X 0,Y 601.346,Z 895.169,A -85,B 0,C 180,E1 -621.261,E2 -621.261} C_VEL
LIN {X 0,Y 601.322,Z 898.306,A -85,B 0,C 180,E1 -622.613,E2 -622.613} C_VEL
LIN {X 0,Y 601.332,Z 900.045,A -85,B 0,C 180,E1 -623.962,E2 -623.962} C_VEL
LIN {X 0,Y 601.321,Z 900.445,A -85,B 0,C 180,E1 -625.307,E2 -625.307} C_VEL
LIN {X 0,Y 601.333,Z 899.522,A -85,B 0,C 180,E1 -626.65,E2 -626.65} C_VEL
LIN {X 0,Y 601.342,Z 897.262,A -85,B 0,C 180,E1 -627.991,E2 -627.991} C_VEL
LIN {X 0,Y 601.339,Z 893.608,A -85,B 0,C 180,E1 -629.33,E2 -629.33} C_VEL
LIN {X 0,Y 601.362,Z 888.468,A -85,B 0,C 180,E1 -630.67,E2 -630.67} C_VEL
LIN {X 0,Y 601.361,Z 883.493,A -85,B 0,C 180,E1 -631.674,E2 -631.674} C_VEL
LIN {X 0,Y 601.372,Z 876.399,A -85,B 0,C 180,E1 -632.847,E2 -632.847} C_VEL
LIN {X 0,Y 601.401,Z 867.65,A -85,B 0,C 180,E1 -634.021,E2 -634.021} C_VEL
LIN {X 0,Y 601.437,Z 858.527,A -85,B 0,C 180,E1 -635.028,E2 -635.028} C_VEL
LIN {X 0,Y 601.484,Z 848.469,A -85,B 0,C 180,E1 -635.952,E2 -635.952} C_VEL
LIN {X 0,Y 601.549,Z 837.563,A -85,B 0,C 180,E1 -636.785,E2 -636.785} C_VEL
LIN {X 0,Y 601.557,Z 825.311,A -85,B 0,C 180,E1 -637.553,E2 -637.553} C_VEL
LIN {X 0,Y 601.63,Z 811.777,A -85,B 0,C 180,E1 -638.227,E2 -638.227} C_VEL
LIN {X 0,Y 601.676,Z 798.635,A -85,B 0,C 180,E1 -638.734,E2 -638.734} C_VEL
LIN {X 0,Y 601.674,Z 784.372,A -85,B 0,C 180,E1 -639.136,E2 -639.136} C_VEL
LIN {X 0,Y 601.714,Z 770.417,A -85,B 0,C 180,E1 -639.39,E2 -639.39} C_VEL
LIN {X 0,Y 601.757,Z 640.559,A -85,B 0,C 180,E1 -640.966,E2 -640.966} C_VEL
LIN {X 0,Y 601.475,Z 638.818,A -85,B 0,C 180,E1 -641.011,E2 -641.011} C_VEL
LIN {X 0,Y 601.515,Z 621.073,A -85,B 0,C 180,E1 -643.668,E2 -643.668} C_VEL
LIN {X 0,Y 601.39,Z 609.702,A -85,B 0,C 180,E1 -645.397,E2 -645.397} C_VEL
LIN {X 0,Y 601.355,Z 609.697,A -85,B 0,C 180,E1 -647.69,E2 -647.69} C_VEL
LIN {X 0,Y 601.426,Z 609.697,A -85,B 0,C 180,E1 -650.522,E2 -650.522} C_VEL
LIN {X 0,Y 601.36,Z 609.696,A -85,B 0,C 180,E1 -653.413,E2 -653.413} C_VEL
LIN {X 0,Y 601.354,Z 609.696,A -85,B 0,C 180,E1 -655.855,E2 -655.855} C_VEL
LIN {X 0,Y 601.421,Z 609.699,A -85,B 0,C 180,E1 -658.785,E2 -658.785} C_VEL
LIN {X 0,Y 601.378,Z 609.693,A -85,B 0,C 180,E1 -661.728,E2 -661.728} C_VEL
LIN {X 0,Y 601.383,Z 609.693,A -85,B 0,C 180,E1 -664.121,E2 -664.121} C_VEL
LIN {X 0,Y 601.393,Z 609.697,A -85,B 0,C 180,E1 -666.584,E2 -666.584} C_VEL
LIN {X 0,Y 601.395,Z 609.692,A -85,B 0,C 180,E1 -669.53,E2 -669.53} C_VEL
LIN {X 0,Y 601.395,Z 609.691,A -85,B 0,C 180,E1 -671.768,E2 -671.768} C_VEL
LIN {X 0,Y 601.402,Z 609.693,A -85,B 0,C 180,E1 -674.532,E2 -674.532} C_VEL
LIN {X 0,Y 601.38,Z 609.698,A -85,B 0,C 180,E1 -677.413,E2 -677.413} C_VEL
LIN {X 0,Y 601.376,Z 609.693,A -85,B 0,C 180,E1 -680.002,E2 -680.002} C_VEL
LIN {X 0,Y 601.39,Z 609.693,A -85,B 0,C 180,E1 -682.624,E2 -682.624} C_VEL
LIN {X 0,Y 601.411,Z 609.697,A -85,B 0,C 180,E1 -685.067,E2 -685.067} C_VEL
LIN {X 0,Y 601.439,Z 609.692,A -85,B 0,C 180,E1 -687.484,E2 -687.484} C_VEL
LIN {X 0,Y 601.405,Z 609.691,A -85,B 0,C 180,E1 -689.856,E2 -689.856} C_VEL
LIN {X 0,Y 601.376,Z 609.694,A -85,B 0,C 180,E1 -692.13,E2 -692.13} C_VEL
LIN {X 0,Y 601.384,Z 609.692,A -85,B 0,C 180,E1 -694.38,E2 -694.38} C_VEL
LIN {X 0,Y 601.379,Z 609.693,A -85,B 0,C 180,E1 -696.588,E2 -696.588} C_VEL
LIN {X 0,Y 601.432,Z 609.697,A -85,B 0,C 180,E1 -699.478,E2 -699.478} C_VEL
LIN {X 0,Y 601.384,Z 609.692,A -85,B 0,C 180,E1 -702.311,E2 -702.311} C_VEL
LIN {X 0,Y 601.397,Z 609.691,A -85,B 0,C 180,E1 -704.408,E2 -704.408} C_VEL
LIN {X 0,Y 601.406,Z 609.694,A -85,B 0,C 180,E1 -707.171,E2 -707.171} C_VEL
LIN {X 0,Y 601.438,Z 609.691,A -85,B 0,C 180,E1 -709.905,E2 -709.905} C_VEL
LIN {X 0,Y 601.403,Z 609.69,A -85,B 0,C 180,E1 -712.614,E2 -712.614} C_VEL
LIN {X 0,Y 601.407,Z 609.693,A -85,B 0,C 180,E1 -715.308,E2 -715.308} C_VEL
LIN {X 0,Y 601.434,Z 609.693,A -85,B 0,C 180,E1 -717.991,E2 -717.991} C_VEL
LIN {X 0,Y 601.448,Z 609.684,A -85,B 0,C 180,E1 -720.669,E2 -720.669} C_VEL
LIN {X 0,Y 601.412,Z 609.692,A -85,B 0,C 180,E1 -723.349,E2 -723.349} C_VEL
LIN {X 0,Y 601.424,Z 609.696,A -85,B 0,C 180,E1 -726.037,E2 -726.037} C_VEL
LIN {X 0,Y 601.417,Z 609.689,A -85,B 0,C 180,E1 -728.738,E2 -728.738} C_VEL
LIN {X 0,Y 601.413,Z 609.691,A -85,B 0,C 180,E1 -731.458,E2 -731.458} C_VEL
LIN {X 0,Y 601.423,Z 609.695,A -85,B 0,C 180,E1 -734.205,E2 -734.205} C_VEL
LIN {X 0,Y 601.432,Z 609.686,A -85,B 0,C 180,E1 -736.986,E2 -736.986} C_VEL
LIN {X 0,Y 601.407,Z 609.695,A -85,B 0,C 180,E1 -739.809,E2 -739.809} C_VEL
LIN {X 0,Y 601.419,Z 609.691,A -85,B 0,C 180,E1 -742.605,E2 -742.605} C_VEL
LIN {X 0,Y 601.405,Z 609.691,A -85,B 0,C 180,E1 -744.878,E2 -744.878} C_VEL
LIN {X 0,Y 601.418,Z 609.688,A -85,B 0,C 180,E1 -747.362,E2 -747.362} C_VEL
LIN {X 0,Y 601.43,Z 609.695,A -85,B 0,C 180,E1 -750.164,E2 -750.164} C_VEL
LIN {X 0,Y 601.428,Z 609.691,A -85,B 0,C 180,E1 -752.716,E2 -752.716} C_VEL
LIN {X 0,Y 601.419,Z 609.689,A -85,B 0,C 180,E1 -755.115,E2 -755.115} C_VEL
LIN {X 0,Y 601.437,Z 609.686,A -85,B 0,C 180,E1 -757.419,E2 -757.419} C_VEL
LIN {X 0,Y 601.413,Z 609.692,A -85,B 0,C 180,E1 -759.995,E2 -759.995} C_VEL
LIN {X 0,Y 601.415,Z 609.696,A -85,B 0,C 180,E1 -762.67,E2 -762.67} C_VEL
LIN {X 0,Y 601.428,Z 609.687,A -85,B 0,C 180,E1 -765.482,E2 -765.482} C_VEL
LIN {X 0,Y 601.431,Z 609.694,A -85,B 0,C 180,E1 -768.406,E2 -768.406} C_VEL
LIN {X 0,Y 601.437,Z 609.686,A -85,B 0,C 180,E1 -771.529,E2 -771.529} C_VEL
LIN {X 0,Y 601.411,Z 609.693,A -85,B 0,C 180,E1 -774.247,E2 -774.247} C_VEL
LIN {X 0,Y 601.429,Z 609.697,A -85,B 0,C 180,E1 -776.686,E2 -776.686} C_VEL
LIN {X 0,Y 601.431,Z 609.693,A -85,B 0,C 180,E1 -779.058,E2 -779.058} C_VEL
LIN {X 0,Y 601.433,Z 609.689,A -85,B 0,C 180,E1 -781.373,E2 -781.373} C_VEL
LIN {X 0,Y 601.421,Z 609.689,A -85,B 0,C 180,E1 -784.131,E2 -784.131} C_VEL
LIN {X 0,Y 601.45,Z 609.792,A -85,B 0,C 180,E1 -785.802,E2 -785.802} C_VEL
LIN {X 0,Y 601.777,Z 613.135,A -85,B 0,C 180,E1 -786.239,E2 -786.239} C_VEL
LIN {X 0,Y 601.69,Z 635.532,A -85,B 0,C 180,E1 -789.04,E2 -789.04} C_VEL
LIN {X 0,Y 601.601,Z 657.921,A -85,B 0,C 180,E1 -791.79,E2 -791.79} C_VEL
LIN {X 0,Y 601.539,Z 676.431,A -85,B 0,C 180,E1 -794.032,E2 -794.032} C_VEL
LIN {X 0,Y 601.848,Z 682.394,A -85,B 0,C 180,E1 -794.116,E2 -794.116} C_VEL
LIN {X 0,Y 601.717,Z 814.975,A -85,B 0,C 180,E1 -795.739,E2 -795.739} C_VEL
LIN {X 0,Y 601.691,Z 829.086,A -85,B 0,C 180,E1 -796.051,E2 -796.051} C_VEL
LIN {X 0,Y 601.666,Z 842.708,A -85,B 0,C 180,E1 -796.49,E2 -796.49} C_VEL
LIN {X 0,Y 601.602,Z 856.63,A -85,B 0,C 180,E1 -797.09,E2 -797.09} C_VEL
LIN {X 0,Y 601.551,Z 869.091,A -85,B 0,C 180,E1 -797.775,E2 -797.775} C_VEL
LIN {X 0,Y 601.504,Z 880.47,A -85,B 0,C 180,E1 -798.543,E2 -798.543} C_VEL
LIN {X 0,Y 601.482,Z 890.93,A -85,B 0,C 180,E1 -799.395,E2 -799.395} C_VEL
LIN {X 0,Y 601.43,Z 901.333,A -85,B 0,C 180,E1 -800.414,E2 -800.414} C_VEL
LIN {X 0,Y 601.407,Z 909.913,A -85,B 0,C 180,E1 -801.431,E2 -801.431} C_VEL
LIN {X 0,Y 601.392,Z 918.113,A -85,B 0,C 180,E1 -802.614,E2 -802.614} C_VEL
LIN {X 0,Y 601.361,Z 923.751,A -85,B 0,C 180,E1 -803.604,E2 -803.604} C_VEL
LIN {X 0,Y 601.354,Z 928.567,A -85,B 0,C 180,E1 -804.635,E2 -804.635} C_VEL
LIN {X 0,Y 601.345,Z 933.441,A -85,B 0,C 180,E1 -805.979,E2 -805.979} C_VEL
LIN {X 0,Y 601.323,Z 936.831,A -85,B 0,C 180,E1 -807.32,E2 -807.32} C_VEL
LIN {X 0,Y 601.342,Z 938.831,A -85,B 0,C 180,E1 -808.661,E2 -808.661} C_VEL
LIN {X 0,Y 601.333,Z 939.5,A -85,B 0,C 180,E1 -810,E2 -810} C_VEL
LIN {X 0,Y 601.342,Z 938.831,A -85,B 0,C 180,E1 -811.339,E2 -811.339} C_VEL
LIN {X 0,Y 601.323,Z 936.832,A -85,B 0,C 180,E1 -812.68,E2 -812.68} C_VEL
LIN {X 0,Y 601.345,Z 933.442,A -85,B 0,C 180,E1 -814.021,E2 -814.021} C_VEL
LIN {X 0,Y 601.354,Z 928.568,A -85,B 0,C 180,E1 -815.365,E2 -815.365} C_VEL
LIN {X 0,Y 601.372,Z 922.623,A -85,B 0,C 180,E1 -816.605,E2 -816.605} C_VEL
LIN {X 0,Y 601.386,Z 915.919,A -85,B 0,C 180,E1 -817.723,E2 -817.723} C_VEL
LIN {X 0,Y 601.411,Z 907.198,A -85,B 0,C 180,E1 -818.907,E2 -818.907} C_VEL
LIN {X 0,Y 601.432,Z 898.082,A -85,B 0,C 180,E1 -819.925,E2 -819.925} C_VEL
LIN {X 0,Y 601.497,Z 887.83,A -85,B 0,C 180,E1 -820.876,E2 -820.876} C_VEL
LIN {X 0,Y 601.534,Z 876.971,A -85,B 0,C 180,E1 -821.712,E2 -821.712} C_VEL
LIN {X 0,Y 601.578,Z 864.776,A -85,B 0,C 180,E1 -822.482,E2 -822.482} C_VEL
LIN {X 0,Y 601.612,Z 853.093,A -85,B 0,C 180,E1 -823.082,E2 -823.082} C_VEL
LIN {X 0,Y 601.65,Z 840.942,A -85,B 0,C 180,E1 -823.578,E2 -823.578} C_VEL
LIN {X 0,Y 601.685,Z 827.044,A -85,B 0,C 180,E1 -824.005,E2 -824.005} C_VEL
LIN {X 0,Y 601.741,Z 812.899,A -85,B 0,C 180,E1 -824.295,E2 -824.295} C_VEL
LIN {X 0,Y 601.682,Z 677.374,A -85,B 0,C 180,E1 -825.95,E2 -825.95} C_VEL
LIN {X 0,Y 601.549,Z 676.342,A -85,B 0,C 180,E1 -825.979,E2 -825.979} C_VEL
LIN {X 0,Y 601.612,Z 652.492,A -85,B 0,C 180,E1 -828.873,E2 -828.873} C_VEL
LIN {X 0,Y 601.695,Z 629.028,A -85,B 0,C 180,E1 -831.768,E2 -831.768} C_VEL
LIN {X 0,Y 601.795,Z 611.692,A -85,B 0,C 180,E1 -833.943,E2 -833.943} C_VEL
LIN {X 0,Y 601.454,Z 609.688,A -85,B 0,C 180,E1 -834.217,E2 -834.217} C_VEL
LIN {X 0,Y 601.452,Z 609.695,A -85,B 0,C 180,E1 -837.111,E2 -837.111} C_VEL
LIN {X 0,Y 601.427,Z 609.695,A -85,B 0,C 180,E1 -839.393,E2 -839.393} C_VEL
LIN {X 0,Y 601.415,Z 609.692,A -85,B 0,C 180,E1 -841.726,E2 -841.726} C_VEL
LIN {X 0,Y 601.433,Z 609.686,A -85,B 0,C 180,E1 -844.118,E2 -844.118} C_VEL
LIN {X 0,Y 601.411,Z 609.689,A -85,B 0,C 180,E1 -846.582,E2 -846.582} C_VEL
LIN {X 0,Y 601.44,Z 609.694,A -85,B 0,C 180,E1 -849.536,E2 -849.536} C_VEL
LIN {X 0,Y 601.431,Z 609.692,A -85,B 0,C 180,E1 -851.765,E2 -851.765} C_VEL
LIN {X 0,Y 601.426,Z 609.687,A -85,B 0,C 180,E1 -854.535,E2 -854.535} C_VEL
LIN {X 0,Y 601.417,Z 609.697,A -85,B 0,C 180,E1 -857.409,E2 -857.409} C_VEL
LIN {X 0,Y 601.442,Z 609.685,A -85,B 0,C 180,E1 -860.464,E2 -860.464} C_VEL
LIN {X 0,Y 601.414,Z 609.695,A -85,B 0,C 180,E1 -863.418,E2 -863.418} C_VEL
LIN {X 0,Y 601.436,Z 609.69,A -85,B 0,C 180,E1 -866.064,E2 -866.064} C_VEL
LIN {X 0,Y 601.444,Z 609.684,A -85,B 0,C 180,E1 -868.542,E2 -868.542} C_VEL
LIN {X 0,Y 601.437,Z 609.689,A -85,B 0,C 180,E1 -871.374,E2 -871.374} C_VEL
LIN {X 0,Y 601.405,Z 609.697,A -85,B 0,C 180,E1 -873.636,E2 -873.636} C_VEL
LIN {X 0,Y 601.421,Z 609.688,A -85,B 0,C 180,E1 -876.59,E2 -876.59} C_VEL
LIN {X 0,Y 601.437,Z 609.689,A -85,B 0,C 180,E1 -879.479,E2 -879.479} C_VEL
LIN {X 0,Y 601.398,Z 609.696,A -85,B 0,C 180,E1 -882.312,E2 -882.312} C_VEL
LIN {X 0,Y 601.414,Z 609.693,A -85,B 0,C 180,E1 -884.409,E2 -884.409} C_VEL
LIN {X 0,Y 601.419,Z 609.688,A -85,B 0,C 180,E1 -887.172,E2 -887.172} C_VEL
LIN {X 0,Y 601.443,Z 609.692,A -85,B 0,C 180,E1 -889.905,E2 -889.905} C_VEL
LIN {X 0,Y 601.407,Z 609.693,A -85,B 0,C 180,E1 -892.615,E2 -892.615} C_VEL
LIN {X 0,Y 601.43,Z 609.686,A -85,B 0,C 180,E1 -895.308,E2 -895.308} C_VEL
LIN {X 0,Y 601.427,Z 609.692,A -85,B 0,C 180,E1 -897.991,E2 -897.991} C_VEL
LIN {X 0,Y 601.443,Z 609.69,A -85,B 0,C 180,E1 -900.67,E2 -900.67} C_VEL
LIN {X 0,Y 601.421,Z 609.688,A -85,B 0,C 180,E1 -903.35,E2 -903.35} C_VEL
LIN {X 0,Y 601.44,Z 609.689,A -85,B 0,C 180,E1 -906.037,E2 -906.037} C_VEL
LIN {X 0,Y 601.412,Z 609.695,A -85,B 0,C 180,E1 -908.738,E2 -908.738} C_VEL
LIN {X 0,Y 601.411,Z 609.689,A -85,B 0,C 180,E1 -911.459,E2 -911.459} C_VEL
LIN {X 0,Y 601.41,Z 609.692,A -85,B 0,C 180,E1 -912.373,E2 -912.373} C_VEL
LIN {X 0,Y 600.741,Z 609.779,A -85,B 0,C 180,E1 -912.933,E2 -912.933} C_VEL
LIN {X 0,Y 597.888,Z 610.134,A -85,B 0,C 180,E1 -913.841,E2 -913.841} C_VEL
LIN {X 0,Y 595.478,Z 610.439,A -85,B 0,C 180,E1 -914.571,E2 -914.571} C_VEL
LIN {X 0,Y 594.441,Z 610.56,A -85,B 0,C 180,E1 -915.134,E2 -915.134} C_VEL
LIN {X 0,Y 594.355,Z 610.569,A -85,B 0,C 180,E1 -915.325,E2 -915.325} C_VEL
LIN {X 0,Y 594.387,Z 610.566,A -85,B 0,C 180,E1 -917.194,E2 -917.194} C_VEL
LIN {X 0,Y 594.374,Z 610.566,A -85,B 0,C 180,E1 -920.054,E2 -920.054} C_VEL
LIN {X 0,Y 594.356,Z 610.575,A -85,B 0,C 180,E1 -922.968,E2 -922.968} C_VEL
LIN {X 0,Y 594.356,Z 610.572,A -85,B 0,C 180,E1 -925.194,E2 -925.194} C_VEL
LIN {X 0,Y 594.344,Z 610.57,A -85,B 0,C 180,E1 -927.519,E2 -927.519} C_VEL
LIN {X 0,Y 594.36,Z 610.566,A -85,B 0,C 180,E1 -929.778,E2 -929.778} C_VEL
LIN {X 0,Y 594.369,Z 610.567,A -85,B 0,C 180,E1 -932.147,E2 -932.147} C_VEL
LIN {X 0,Y 594.378,Z 610.569,A -85,B 0,C 180,E1 -934.581,E2 -934.581} C_VEL
LIN {X 0,Y 594.385,Z 610.566,A -85,B 0,C 180,E1 -937.608,E2 -937.608} C_VEL
LIN {X 0,Y 594.36,Z 610.569,A -85,B 0,C 180,E1 -940.568,E2 -940.568} C_VEL
LIN {X 0,Y 594.349,Z 610.577,A -85,B 0,C 180,E1 -943.302,E2 -943.302} C_VEL
LIN {X 0,Y 594.346,Z 610.569,A -85,B 0,C 180,E1 -946.163,E2 -946.163} C_VEL
LIN {X 0,Y 594.373,Z 610.576,A -85,B 0,C 180,E1 -949.179,E2 -949.179} C_VEL
LIN {X 0,Y 594.369,Z 610.567,A -85,B 0,C 180,E1 -952.058,E2 -952.058} C_VEL
LIN {X 0,Y 594.332,Z 610.572,A -85,B 0,C 180,E1 -954.68,E2 -954.68} C_VEL
LIN {X 0,Y 594.377,Z 610.571,A -85,B 0,C 180,E1 -957.09,E2 -957.09} C_VEL
LIN {X 0,Y 594.368,Z 610.574,A -85,B 0,C 180,E1 -959.676,E2 -959.676} C_VEL
LIN {X 0,Y 594.339,Z 610.577,A -85,B 0,C 180,E1 -961.771,E2 -961.771} C_VEL
LIN {X 0,Y 594.354,Z 610.696,A -85,B 0,C 180,E1 -964.595,E2 -964.595} C_VEL
LIN {X 0,Y 594.559,Z 616.927,A -85,B 0,C 180,E1 -965.561,E2 -965.561} C_VEL
LIN {X 0,Y 594.508,Z 635.063,A -85,B 0,C 180,E1 -968.32,E2 -968.32} C_VEL
LIN {X 0,Y 594.499,Z 638.914,A -85,B 0,C 180,E1 -968.901,E2 -968.901} C_VEL
LIN {X 0,Y 595.021,Z 643.634,A -85,B 0,C 180,E1 -968.977,E2 -968.977} C_VEL
LIN {X 0,Y 594.823,Z 774.636,A -85,B 0,C 180,E1 -970.591,E2 -970.591} C_VEL
LIN {X 0,Y 594.803,Z 789.373,A -85,B 0,C 180,E1 -970.911,E2 -970.911} C_VEL
LIN {X 0,Y 594.75,Z 802.984,A -85,B 0,C 180,E1 -971.347,E2 -971.347} C_VEL
LIN {X 0,Y 594.644,Z 816.525,A -85,B 0,C 180,E1 -971.926,E2 -971.926} C_VEL
LIN {X 0,Y 594.585,Z 829.459,A -85,B 0,C 180,E1 -972.635,E2 -972.635} C_VEL
LIN {X 0,Y 594.507,Z 841.227,A -85,B 0,C 180,E1 -973.433,E2 -973.433} C_VEL
LIN {X 0,Y 594.459,Z 852.876,A -85,B 0,C 180,E1 -974.398,E2 -974.398} C_VEL
LIN {X 0,Y 594.382,Z 863.254,A -85,B 0,C 180,E1 -975.448,E2 -975.448} C_VEL
LIN {X 0,Y 594.342,Z 871.805,A -85,B 0,C 180,E1 -976.494,E2 -976.494} C_VEL
LIN {X 0,Y 594.292,Z 879.938,A -85,B 0,C 180,E1 -977.71,E2 -977.71} C_VEL
LIN {X 0,Y 594.252,Z 886.823,A -85,B 0,C 180,E1 -978.997,E2 -978.997} C_VEL
LIN {X 0,Y 594.259,Z 891.579,A -85,B 0,C 180,E1 -980.126,E2 -980.126} C_VEL
LIN {X 0,Y 594.246,Z 895,A -85,B 0,C 180,E1 -981.156,E2 -981.156} C_VEL
LIN {X 0,Y 594.247,Z 898.208,A -85,B 0,C 180,E1 -982.525,E2 -982.525} C_VEL
LIN {X 0,Y 594.237,Z 900.004,A -85,B 0,C 180,E1 -983.89,E2 -983.89} C_VEL
LIN {X 0,Y 594.22,Z 900.459,A -85,B 0,C 180,E1 -985.251,E2 -985.251} C_VEL
LIN {X 0,Y 594.253,Z 899.59,A -85,B 0,C 180,E1 -986.61,E2 -986.61} C_VEL
LIN {X 0,Y 594.241,Z 897.387,A -85,B 0,C 180,E1 -987.967,E2 -987.967} C_VEL
LIN {X 0,Y 594.24,Z 893.793,A -85,B 0,C 180,E1 -989.322,E2 -989.322} C_VEL
LIN {X 0,Y 594.267,Z 888.717,A -85,B 0,C 180,E1 -990.678,E2 -990.678} C_VEL
LIN {X 0,Y 594.284,Z 883.809,A -85,B 0,C 180,E1 -991.694,E2 -991.694} C_VEL
LIN {X 0,Y 594.303,Z 876.789,A -85,B 0,C 180,E1 -992.881,E2 -992.881} C_VEL
LIN {X 0,Y 594.348,Z 868.124,A -85,B 0,C 180,E1 -994.069,E2 -994.069} C_VEL
LIN {X 0,Y 594.387,Z 859.093,A -85,B 0,C 180,E1 -995.088,E2 -995.088} C_VEL
LIN {X 0,Y 594.494,Z 848.163,A -85,B 0,C 180,E1 -996.108,E2 -996.108} C_VEL
LIN {X 0,Y 594.579,Z 836.291,A -85,B 0,C 180,E1 -997.011,E2 -997.011} C_VEL
LIN {X 0,Y 594.609,Z 823.308,A -85,B 0,C 180,E1 -997.812,E2 -997.812} C_VEL
LIN {X 0,Y 594.682,Z 811.201,A -85,B 0,C 180,E1 -998.41,E2 -998.41} C_VEL
LIN {X 0,Y 594.79,Z 797.865,A -85,B 0,C 180,E1 -998.922,E2 -998.922} C_VEL
LIN {X 0,Y 594.804,Z 784.181,A -85,B 0,C 180,E1 -999.307,E2 -999.307} C_VEL
LIN {X 0,Y 594.845,Z 770.105,A -85,B 0,C 180,E1 -999.564,E2 -999.564} C_VEL
LIN {X 0,Y 594.959,Z 641.837,A -85,B 0,C 180,E1 -1001.137,E2 -1001.137} C_VEL
LIN {X 0,Y 594.463,Z 638.829,A -85,B 0,C 180,E1 -1001.203,E2 -1001.203} C_VEL
LIN {X 0,Y 594.524,Z 622.508,A -85,B 0,C 180,E1 -1003.676,E2 -1003.676} C_VEL
LIN {X 0,Y 594.565,Z 612.244,A -85,B 0,C 180,E1 -1005.249,E2 -1005.249} C_VEL
LIN {X 0,Y 594.34,Z 610.575,A -85,B 0,C 180,E1 -1005.518,E2 -1005.518} C_VEL
LIN {X 0,Y 594.317,Z 610.575,A -85,B 0,C 180,E1 -1007.906,E2 -1007.906} C_VEL
LIN {X 0,Y 594.404,Z 610.571,A -85,B 0,C 180,E1 -1010.776,E2 -1010.776} C_VEL
LIN {X 0,Y 594.344,Z 610.57,A -85,B 0,C 180,E1 -1013.706,E2 -1013.706} C_VEL
LIN {X 0,Y 594.346,Z 610.58,A -85,B 0,C 180,E1 -1016.702,E2 -1016.702} C_VEL
LIN {X 0,Y 594.373,Z 610.573,A -85,B 0,C 180,E1 -1018.999,E2 -1018.999} C_VEL
LIN {X 0,Y 594.354,Z 610.569,A -85,B 0,C 180,E1 -1021.638,E2 -1021.638} C_VEL
LIN {X 0,Y 594.366,Z 610.573,A -85,B 0,C 180,E1 -1024.581,E2 -1024.581} C_VEL
LIN {X 0,Y 594.357,Z 610.569,A -85,B 0,C 180,E1 -1027.604,E2 -1027.604} C_VEL
LIN {X 0,Y 594.336,Z 610.57,A -85,B 0,C 180,E1 -1029.769,E2 -1029.769} C_VEL
LIN {X 0,Y 594.334,Z 610.572,A -85,B 0,C 180,E1 -1032.379,E2 -1032.379} C_VEL
LIN {X 0,Y 594.341,Z 610.578,A -85,B 0,C 180,E1 -1035.194,E2 -1035.194} C_VEL
LIN {X 0,Y 594.344,Z 610.569,A -85,B 0,C 180,E1 -1038.156,E2 -1038.156} C_VEL
LIN {X 0,Y 594.349,Z 610.569,A -85,B 0,C 180,E1 -1040.317,E2 -1040.317} C_VEL
LIN {X 0,Y 594.354,Z 610.573,A -85,B 0,C 180,E1 -1042.911,E2 -1042.911} C_VEL
LIN {X 0,Y 594.367,Z 610.568,A -85,B 0,C 180,E1 -1045.864,E2 -1045.864} C_VEL
LIN {X 0,Y 594.359,Z 610.569,A -85,B 0,C 180,E1 -1048.649,E2 -1048.649} C_VEL
LIN {X 0,Y 594.381,Z 610.57,A -85,B 0,C 180,E1 -1051.043,E2 -1051.043} C_VEL
LIN {X 0,Y 594.341,Z 610.57,A -85,B 0,C 180,E1 -1054.054,E2 -1054.054} C_VEL
LIN {X 0,Y 594.368,Z 610.566,A -85,B 0,C 180,E1 -1056.295,E2 -1056.295} C_VEL
LIN {X 0,Y 594.403,Z 610.569,A -85,B 0,C 180,E1 -1059.224,E2 -1059.224} C_VEL
LIN {X 0,Y 594.347,Z 610.57,A -85,B 0,C 180,E1 -1062.095,E2 -1062.095} C_VEL
LIN {X 0,Y 594.356,Z 610.569,A -85,B 0,C 180,E1 -1064.219,E2 -1064.219} C_VEL
LIN {X 0,Y 594.374,Z 610.566,A -85,B 0,C 180,E1 -1066.321,E2 -1066.321} C_VEL
LIN {X 0,Y 594.353,Z 610.57,A -85,B 0,C 180,E1 -1069.094,E2 -1069.094} C_VEL
LIN {X 0,Y 594.414,Z 610.568,A -85,B 0,C 180,E1 -1071.843,E2 -1071.843} C_VEL
LIN {X 0,Y 594.38,Z 610.565,A -85,B 0,C 180,E1 -1074.572,E2 -1074.572} C_VEL
LIN {X 0,Y 594.394,Z 610.566,A -85,B 0,C 180,E1 -1077.289,E2 -1077.289} C_VEL
LIN {X 0,Y 594.42,Z 610.567,A -85,B 0,C 180,E1 -1080,E2 -1080} C_VEL
LIN {X 0,Y 594.411,Z 610.561,A -85,B 0,C 180,E1 -1082.711,E2 -1082.711} C_VEL
LIN {X 0,Y 594.382,Z 610.568,A -85,B 0,C 180,E1 -1085.428,E2 -1085.428} C_VEL
LIN {X 0,Y 594.416,Z 610.567,A -85,B 0,C 180,E1 -1088.157,E2 -1088.157} C_VEL
LIN {X 0,Y 594.394,Z 610.563,A -85,B 0,C 180,E1 -1091.074,E2 -1091.074} C_VEL
LIN {X 0,Y 594.381,Z 610.57,A -85,B 0,C 180,E1 -1093.679,E2 -1093.679} C_VEL
LIN {X 0,Y 594.399,Z 610.564,A -85,B 0,C 180,E1 -1096.72,E2 -1096.72} C_VEL
LIN {X 0,Y 594.37,Z 610.566,A -85,B 0,C 180,E1 -1099.334,E2 -1099.334} C_VEL
LIN {X 0,Y 594.368,Z 610.568,A -85,B 0,C 180,E1 -1101.503,E2 -1101.503} C_VEL
LIN {X 0,Y 594.392,Z 610.57,A -85,B 0,C 180,E1 -1104.446,E2 -1104.446} C_VEL
LIN {X 0,Y 594.388,Z 610.567,A -85,B 0,C 180,E1 -1106.699,E2 -1106.699} C_VEL
LIN {X 0,Y 594.385,Z 610.565,A -85,B 0,C 180,E1 -1108.998,E2 -1108.998} C_VEL
LIN {X 0,Y 594.387,Z 610.565,A -85,B 0,C 180,E1 -1111.644,E2 -1111.644} C_VEL
LIN {X 0,Y 594.4,Z 610.57,A -85,B 0,C 180,E1 -1114.579,E2 -1114.579} C_VEL
LIN {X 0,Y 594.392,Z 610.564,A -85,B 0,C 180,E1 -1117.608,E2 -1117.608} C_VEL
LIN {X 0,Y 594.373,Z 610.575,A -85,B 0,C 180,E1 -1120.567,E2 -1120.567} C_VEL
LIN {X 0,Y 594.369,Z 610.567,A -85,B 0,C 180,E1 -1123.299,E2 -1123.299} C_VEL
LIN {X 0,Y 594.37,Z 610.57,A -85,B 0,C 180,E1 -1126.16,E2 -1126.16} C_VEL
LIN {X 0,Y 594.388,Z 610.574,A -85,B 0,C 180,E1 -1128.537,E2 -1128.537} C_VEL
LIN {X 0,Y 594.386,Z 610.566,A -85,B 0,C 180,E1 -1131.296,E2 -1131.296} C_VEL
LIN {X 0,Y 594.397,Z 610.563,A -85,B 0,C 180,E1 -1133.759,E2 -1133.759} C_VEL
LIN {X 0,Y 594.382,Z 610.568,A -85,B 0,C 180,E1 -1136.239,E2 -1136.239} C_VEL
LIN {X 0,Y 594.393,Z 610.572,A -85,B 0,C 180,E1 -1138.651,E2 -1138.651} C_VEL
LIN {X 0,Y 594.386,Z 610.572,A -85,B 0,C 180,E1 -1141.042,E2 -1141.042} C_VEL
LIN {X 0,Y 594.394,Z 610.565,A -85,B 0,C 180,E1 -1143.976,E2 -1143.976} C_VEL
LIN {X 0,Y 594.393,Z 610.622,A -85,B 0,C 180,E1 -1145.602,E2 -1145.602} C_VEL
LIN {X 0,Y 594.932,Z 614.58,A -85,B 0,C 180,E1 -1146.134,E2 -1146.134} C_VEL
LIN {X 0,Y 594.773,Z 637.123,A -85,B 0,C 180,E1 -1148.985,E2 -1148.985} C_VEL
LIN {X 0,Y 594.663,Z 659.365,A -85,B 0,C 180,E1 -1151.748,E2 -1151.748} C_VEL
LIN {X 0,Y 594.546,Z 676.431,A -85,B 0,C 180,E1 -1153.839,E2 -1153.839} C_VEL
LIN {X 0,Y 595.008,Z 680.605,A -85,B 0,C 180,E1 -1153.906,E2 -1153.906} C_VEL
LIN {X 0,Y 594.857,Z 814.879,A -85,B 0,C 180,E1 -1155.569,E2 -1155.569} C_VEL
LIN {X 0,Y 594.81,Z 829.176,A -85,B 0,C 180,E1 -1155.889,E2 -1155.889} C_VEL
LIN {X 0,Y 594.734,Z 842.71,A -85,B 0,C 180,E1 -1156.329,E2 -1156.329} C_VEL
LIN {X 0,Y 594.646,Z 856.632,A -85,B 0,C 180,E1 -1156.936,E2 -1156.936} C_VEL
LIN {X 0,Y 594.6,Z 869.092,A -85,B 0,C 180,E1 -1157.629,E2 -1157.629} C_VEL
LIN {X 0,Y 594.514,Z 880.472,A -85,B 0,C 180,E1 -1158.407,E2 -1158.407} C_VEL
LIN {X 0,Y 594.474,Z 890.931,A -85,B 0,C 180,E1 -1159.269,E2 -1159.269} C_VEL
LIN {X 0,Y 594.39,Z 901.333,A -85,B 0,C 180,E1 -1160.3,E2 -1160.3} C_VEL
LIN {X 0,Y 594.355,Z 909.913,A -85,B 0,C 180,E1 -1161.329,E2 -1161.329} C_VEL
LIN {X 0,Y 594.314,Z 918.114,A -85,B 0,C 180,E1 -1162.526,E2 -1162.526} C_VEL
LIN {X 0,Y 594.27,Z 924.233,A -85,B 0,C 180,E1 -1163.619,E2 -1163.619} C_VEL
LIN {X 0,Y 594.246,Z 929.961,A -85,B 0,C 180,E1 -1164.911,E2 -1164.911} C_VEL
LIN {X 0,Y 594.26,Z 933.441,A -85,B 0,C 180,E1 -1165.931,E2 -1165.931} C_VEL
LIN {X 0,Y 594.224,Z 936.831,A -85,B 0,C 180,E1 -1167.288,E2 -1167.288} C_VEL
LIN {X 0,Y 594.242,Z 938.831,A -85,B 0,C 180,E1 -1168.645,E2 -1168.645} C_VEL
LIN {X 0,Y 594.234,Z 939.5,A -85,B 0,C 180,E1 -1170,E2 -1170} C_VEL
LIN {X 0,Y 594.242,Z 938.831,A -85,B 0,C 180,E1 -1171.355,E2 -1171.355} C_VEL
LIN {X 0,Y 594.224,Z 936.832,A -85,B 0,C 180,E1 -1172.712,E2 -1172.712} C_VEL
LIN {X 0,Y 594.26,Z 933.442,A -85,B 0,C 180,E1 -1174.069,E2 -1174.069} C_VEL
LIN {X 0,Y 594.274,Z 928.568,A -85,B 0,C 180,E1 -1175.429,E2 -1175.429} C_VEL
LIN {X 0,Y 594.299,Z 923.033,A -85,B 0,C 180,E1 -1176.607,E2 -1176.607} C_VEL
LIN {X 0,Y 594.316,Z 915.919,A -85,B 0,C 180,E1 -1177.816,E2 -1177.816} C_VEL
LIN {X 0,Y 594.369,Z 907.199,A -85,B 0,C 180,E1 -1179.014,E2 -1179.014} C_VEL
LIN {X 0,Y 594.4,Z 898.082,A -85,B 0,C 180,E1 -1180.044,E2 -1180.044} C_VEL
LIN {X 0,Y 594.478,Z 887.702,A -85,B 0,C 180,E1 -1181.018,E2 -1181.018} C_VEL
LIN {X 0,Y 594.568,Z 875.705,A -85,B 0,C 180,E1 -1181.938,E2 -1181.938} C_VEL
LIN {X 0,Y 594.619,Z 863.211,A -85,B 0,C 180,E1 -1182.717,E2 -1182.717} C_VEL
LIN {X 0,Y 594.694,Z 851.129,A -85,B 0,C 180,E1 -1183.323,E2 -1183.323} C_VEL
LIN {X 0,Y 594.782,Z 837.201,A -85,B 0,C 180,E1 -1183.866,E2 -1183.866} C_VEL
LIN {X 0,Y 594.816,Z 823.288,A -85,B 0,C 180,E1 -1184.259,E2 -1184.259} C_VEL
LIN {X 0,Y 594.873,Z 809.122,A -85,B 0,C 180,E1 -1184.518,E2 -1184.518} C_VEL
LIN {X 0,Y 594.878,Z 678.382,A -85,B 0,C 180,E1 -1186.124,E2 -1186.124} C_VEL
LIN {X 0,Y 594.557,Z 676.342,A -85,B 0,C 180,E1 -1186.172,E2 -1186.172} C_VEL
LIN {X 0,Y 594.677,Z 654.214,A -85,B 0,C 180,E1 -1188.888,E2 -1188.888} C_VEL
LIN {X 0,Y 594.815,Z 630.473,A -85,B 0,C 180,E1 -1191.85,E2 -1191.85} C_VEL
LIN {X 0,Y 594.9,Z 613.136,A -85,B 0,C 180,E1 -1194.053,E2 -1194.053} C_VEL
LIN {X 0,Y 594.392,Z 610.571,A -85,B 0,C 180,E1 -1194.434,E2 -1194.434} C_VEL
LIN {X 0,Y 594.388,Z 610.569,A -85,B 0,C 180,E1 -1196.699,E2 -1196.699} C_VEL
LIN {X 0,Y 594.384,Z 610.573,A -85,B 0,C 180,E1 -1198.998,E2 -1198.998} C_VEL
LIN {X 0,Y 594.394,Z 610.567,A -85,B 0,C 180,E1 -1201.645,E2 -1201.645} C_VEL
LIN {X 0,Y 594.399,Z 610.563,A -85,B 0,C 180,E1 -1204.579,E2 -1204.579} C_VEL
LIN {X 0,Y 594.386,Z 610.57,A -85,B 0,C 180,E1 -1207.087,E2 -1207.087} C_VEL
LIN {X 0,Y 594.377,Z 610.569,A -85,B 0,C 180,E1 -1209.774,E2 -1209.774} C_VEL
LIN {X 0,Y 594.373,Z 610.566,A -85,B 0,C 180,E1 -1212.375,E2 -1212.375} C_VEL
LIN {X 0,Y 594.365,Z 610.572,A -85,B 0,C 180,E1 -1215.191,E2 -1215.191} C_VEL
LIN {X 0,Y 594.385,Z 610.566,A -85,B 0,C 180,E1 -1218.152,E2 -1218.152} C_VEL
LIN {X 0,Y 594.389,Z 610.568,A -85,B 0,C 180,E1 -1221.195,E2 -1221.195} C_VEL
LIN {X 0,Y 594.397,Z 610.572,A -85,B 0,C 180,E1 -1223.759,E2 -1223.759} C_VEL
LIN {X 0,Y 594.383,Z 610.567,A -85,B 0,C 180,E1 -1226.239,E2 -1226.239} C_VEL
LIN {X 0,Y 594.393,Z 610.562,A -85,B 0,C 180,E1 -1228.651,E2 -1228.651} C_VEL
LIN {X 0,Y 594.386,Z 610.564,A -85,B 0,C 180,E1 -1231.042,E2 -1231.042} C_VEL
LIN {X 0,Y 594.385,Z 610.573,A -85,B 0,C 180,E1 -1233.978,E2 -1233.978} C_VEL
LIN {X 0,Y 594.393,Z 610.567,A -85,B 0,C 180,E1 -1236.296,E2 -1236.296} C_VEL
LIN {X 0,Y 594.409,Z 610.562,A -85,B 0,C 180,E1 -1239.225,E2 -1239.225} C_VEL
LIN {X 0,Y 594.381,Z 610.574,A -85,B 0,C 180,E1 -1242.096,E2 -1242.096} C_VEL
LIN {X 0,Y 594.369,Z 610.574,A -85,B 0,C 180,E1 -1244.219,E2 -1244.219} C_VEL
LIN {X 0,Y 594.382,Z 610.571,A -85,B 0,C 180,E1 -1246.321,E2 -1246.321} C_VEL
LIN {X 0,Y 594.38,Z 610.565,A -85,B 0,C 180,E1 -1249.095,E2 -1249.095} C_VEL
LIN {X 0,Y 594.416,Z 610.565,A -85,B 0,C 180,E1 -1251.843,E2 -1251.843} C_VEL
LIN {X 0,Y 594.384,Z 610.569,A -85,B 0,C 180,E1 -1254.572,E2 -1254.572} C_VEL
LIN {X 0,Y 594.413,Z 610.561,A -85,B 0,C 180,E1 -1257.289,E2 -1257.289} C_VEL
LIN {X 0,Y 594.415,Z 610.565,A -85,B 0,C 180,E1 -1260,E2 -1260} C_VEL
LIN {X 0,Y 594.403,Z 610.567,A -85,B 0,C 180,E1 -1262.711,E2 -1262.711} C_VEL
LIN {X 0,Y 594.388,Z 610.563,A -85,B 0,C 180,E1 -1265.428,E2 -1265.428} C_VEL
LIN {X 0,Y 594.418,Z 610.565,A -85,B 0,C 180,E1 -1268.157,E2 -1268.157} C_VEL
LIN {X 0,Y 594.389,Z 610.566,A -85,B 0,C 180,E1 -1271.072,E2 -1271.072} C_VEL
LIN {X 0,Y 594.377,Z 610.565,A -85,B 0,C 180,E1 -1273.679,E2 -1273.679} C_VEL
LIN {X 0,Y 594.355,Z 610.569,A -85,B 0,C 180,E1 -1275.325,E2 -1275.325} C_VEL
LIN {X 0,Y 593.681,Z 610.653,A -85,B 0,C 180,E1 -1275.891,E2 -1275.891} C_VEL
LIN {X 0,Y 590.816,Z 611.017,A -85,B 0,C 180,E1 -1276.809,E2 -1276.809} C_VEL
LIN {X 0,Y 588.407,Z 611.314,A -85,B 0,C 180,E1 -1277.548,E2 -1277.548} C_VEL
LIN {X 0,Y 587.386,Z 611.438,A -85,B 0,C 180,E1 -1278.118,E2 -1278.118} C_VEL
LIN {X 0,Y 587.309,Z 611.448,A -85,B 0,C 180,E1 -1278.311,E2 -1278.311} C_VEL
LIN {X 0,Y 587.334,Z 611.448,A -85,B 0,C 180,E1 -1281.038,E2 -1281.038} C_VEL
LIN {X 0,Y 587.314,Z 611.448,A -85,B 0,C 180,E1 -1283.259,E2 -1283.259} C_VEL
LIN {X 0,Y 587.319,Z 611.445,A -85,B 0,C 180,E1 -1285.518,E2 -1285.518} C_VEL
LIN {X 0,Y 587.307,Z 611.445,A -85,B 0,C 180,E1 -1287.82,E2 -1287.82} C_VEL
LIN {X 0,Y 587.327,Z 611.446,A -85,B 0,C 180,E1 -1290.508,E2 -1290.508} C_VEL
LIN {X 0,Y 587.339,Z 611.45,A -85,B 0,C 180,E1 -1293.111,E2 -1293.111} C_VEL
LIN {X 0,Y 587.29,Z 611.448,A -85,B 0,C 180,E1 -1295.901,E2 -1295.901} C_VEL
LIN {X 0,Y 587.319,Z 611.447,A -85,B 0,C 180,E1 -1298.481,E2 -1298.481} C_VEL
LIN {X 0,Y 587.332,Z 611.453,A -85,B 0,C 180,E1 -1301.158,E2 -1301.158} C_VEL
LIN {X 0,Y 587.305,Z 611.446,A -85,B 0,C 180,E1 -1304.111,E2 -1304.111} C_VEL
LIN {X 0,Y 587.294,Z 611.455,A -85,B 0,C 180,E1 -1306.992,E2 -1306.992} C_VEL
LIN {X 0,Y 587.304,Z 611.45,A -85,B 0,C 180,E1 -1309.745,E2 -1309.745} C_VEL
LIN {X 0,Y 587.338,Z 611.443,A -85,B 0,C 180,E1 -1312.392,E2 -1312.392} C_VEL
LIN {X 0,Y 587.313,Z 611.449,A -85,B 0,C 180,E1 -1314.943,E2 -1314.943} C_VEL
LIN {X 0,Y 587.334,Z 611.452,A -85,B 0,C 180,E1 -1317.421,E2 -1317.421} C_VEL
LIN {X 0,Y 587.312,Z 611.451,A -85,B 0,C 180,E1 -1319.829,E2 -1319.829} C_VEL
LIN {X 0,Y 587.301,Z 611.448,A -85,B 0,C 180,E1 -1322.318,E2 -1322.318} C_VEL
LIN {X 0,Y 587.338,Z 611.615,A -85,B 0,C 180,E1 -1324.484,E2 -1324.484} C_VEL
LIN {X 0,Y 587.607,Z 617.22,A -85,B 0,C 180,E1 -1325.367,E2 -1325.367} C_VEL
LIN {X 0,Y 587.516,Z 635.836,A -85,B 0,C 180,E1 -1328.233,E2 -1328.233} C_VEL
LIN {X 0,Y 587.483,Z 638.842,A -85,B 0,C 180,E1 -1328.691,E2 -1328.691} C_VEL
LIN {X 0,Y 588.217,Z 644.26,A -85,B 0,C 180,E1 -1328.794,E2 -1328.794} C_VEL
LIN {X 0,Y 587.96,Z 774.939,A -85,B 0,C 180,E1 -1330.424,E2 -1330.424} C_VEL
LIN {X 0,Y 587.921,Z 789.243,A -85,B 0,C 180,E1 -1330.739,E2 -1330.739} C_VEL
LIN {X 0,Y 587.828,Z 802.599,A -85,B 0,C 180,E1 -1331.167,E2 -1331.167} C_VEL
LIN {X 0,Y 587.757,Z 815.27,A -85,B 0,C 180,E1 -1331.707,E2 -1331.707} C_VEL
LIN {X 0,Y 587.632,Z 828.449,A -85,B 0,C 180,E1 -1332.423,E2 -1332.423} C_VEL
LIN {X 0,Y 587.536,Z 840.442,A -85,B 0,C 180,E1 -1333.234,E2 -1333.234} C_VEL
LIN {X 0,Y 587.453,Z 852.183,A -85,B 0,C 180,E1 -1334.207,E2 -1334.207} C_VEL
LIN {X 0,Y 587.358,Z 862.718,A -85,B 0,C 180,E1 -1335.27,E2 -1335.27} C_VEL
LIN {X 0,Y 587.284,Z 871.363,A -85,B 0,C 180,E1 -1336.329,E2 -1336.329} C_VEL
LIN {X 0,Y 587.219,Z 879.579,A -85,B 0,C 180,E1 -1337.559,E2 -1337.559} C_VEL
LIN {X 0,Y 587.203,Z 885.347,A -85,B 0,C 180,E1 -1338.61,E2 -1338.61} C_VEL
LIN {X 0,Y 587.177,Z 890.009,A -85,B 0,C 180,E1 -1339.657,E2 -1339.657} C_VEL
LIN {X 0,Y 587.151,Z 894.817,A -85,B 0,C 180,E1 -1341.048,E2 -1341.048} C_VEL
LIN {X 0,Y 587.146,Z 898.104,A -85,B 0,C 180,E1 -1342.434,E2 -1342.434} C_VEL
LIN {X 0,Y 587.148,Z 899.962,A -85,B 0,C 180,E1 -1343.816,E2 -1343.816} C_VEL
LIN {X 0,Y 587.12,Z 900.472,A -85,B 0,C 180,E1 -1345.193,E2 -1345.193} C_VEL
LIN {X 0,Y 587.176,Z 899.658,A -85,B 0,C 180,E1 -1346.569,E2 -1346.569} C_VEL
LIN {X 0,Y 587.139,Z 897.513,A -85,B 0,C 180,E1 -1347.942,E2 -1347.942} C_VEL
LIN {X 0,Y 587.142,Z 893.978,A -85,B 0,C 180,E1 -1349.314,E2 -1349.314} C_VEL
LIN {X 0,Y 587.173,Z 888.965,A -85,B 0,C 180,E1 -1350.686,E2 -1350.686} C_VEL
LIN {X 0,Y 587.206,Z 882.322,A -85,B 0,C 180,E1 -1352.058,E2 -1352.058} C_VEL
LIN {X 0,Y 587.262,Z 874.943,A -85,B 0,C 180,E1 -1353.259,E2 -1353.259} C_VEL
LIN {X 0,Y 587.311,Z 867.249,A -85,B 0,C 180,E1 -1354.289,E2 -1354.289} C_VEL
LIN {X 0,Y 587.4,Z 858.032,A -85,B 0,C 180,E1 -1355.321,E2 -1355.321} C_VEL
LIN {X 0,Y 587.503,Z 847.673,A -85,B 0,C 180,E1 -1356.281,E2 -1356.281} C_VEL
LIN {X 0,Y 587.594,Z 836.685,A -85,B 0,C 180,E1 -1357.128,E2 -1357.128} C_VEL
LIN {X 0,Y 587.66,Z 824.39,A -85,B 0,C 180,E1 -1357.905,E2 -1357.905} C_VEL
LIN {X 0,Y 587.758,Z 810.622,A -85,B 0,C 180,E1 -1358.596,E2 -1358.596} C_VEL
LIN {X 0,Y 587.862,Z 797.108,A -85,B 0,C 180,E1 -1359.114,E2 -1359.114} C_VEL
LIN {X 0,Y 587.939,Z 783.091,A -85,B 0,C 180,E1 -1359.504,E2 -1359.504} C_VEL
LIN {X 0,Y 587.98,Z 769.795,A -85,B 0,C 180,E1 -1359.742,E2 -1359.742} C_VEL
LIN {X 0,Y 588.065,Z 642.169,A -85,B 0,C 180,E1 -1361.327,E2 -1361.327} C_VEL
LIN {X 0,Y 587.476,Z 638.816,A -85,B 0,C 180,E1 -1361.403,E2 -1361.403} C_VEL
LIN {X 0,Y 587.569,Z 621.757,A -85,B 0,C 180,E1 -1364.021,E2 -1364.021} C_VEL
LIN {X 0,Y 587.509,Z 612.665,A -85,B 0,C 180,E1 -1365.436,E2 -1365.436} C_VEL
LIN {X 0,Y 587.311,Z 611.452,A -85,B 0,C 180,E1 -1365.664,E2 -1365.664} C_VEL
LIN {X 0,Y 587.277,Z 611.455,A -85,B 0,C 180,E1 -1368.128,E2 -1368.128} C_VEL
LIN {X 0,Y 587.337,Z 611.447,A -85,B 0,C 180,E1 -1371.037,E2 -1371.037} C_VEL
LIN {X 0,Y 587.289,Z 611.45,A -85,B 0,C 180,E1 -1374.009,E2 -1374.009} C_VEL
LIN {X 0,Y 587.295,Z 611.453,A -85,B 0,C 180,E1 -1377.048,E2 -1377.048} C_VEL
LIN {X 0,Y 587.304,Z 611.448,A -85,B 0,C 180,E1 -1379.382,E2 -1379.382} C_VEL
LIN {X 0,Y 587.318,Z 611.445,A -85,B 0,C 180,E1 -1381.831,E2 -1381.831} C_VEL
LIN {X 0,Y 587.319,Z 611.447,A -85,B 0,C 180,E1 -1384.343,E2 -1384.343} C_VEL
LIN {X 0,Y 587.312,Z 611.446,A -85,B 0,C 180,E1 -1387.61,E2 -1387.61} C_VEL
LIN {X 0,Y 587.293,Z 611.447,A -85,B 0,C 180,E1 -1390.256,E2 -1390.256} C_VEL
LIN {X 0,Y 587.292,Z 611.457,A -85,B 0,C 180,E1 -1393.115,E2 -1393.115} C_VEL
LIN {X 0,Y 587.299,Z 611.447,A -85,B 0,C 180,E1 -1396.047,E2 -1396.047} C_VEL
LIN {X 0,Y 587.305,Z 611.454,A -85,B 0,C 180,E1 -1398.929,E2 -1398.929} C_VEL
LIN {X 0,Y 587.311,Z 611.448,A -85,B 0,C 180,E1 -1401.519,E2 -1401.519} C_VEL
LIN {X 0,Y 587.28,Z 611.448,A -85,B 0,C 180,E1 -1404.099,E2 -1404.099} C_VEL
LIN {X 0,Y 587.336,Z 611.447,A -85,B 0,C 180,E1 -1406.889,E2 -1406.889} C_VEL
LIN {X 0,Y 587.321,Z 611.45,A -85,B 0,C 180,E1 -1409.493,E2 -1409.493} C_VEL
LIN {X 0,Y 587.304,Z 611.446,A -85,B 0,C 180,E1 -1412.18,E2 -1412.18} C_VEL
LIN {X 0,Y 587.297,Z 611.447,A -85,B 0,C 180,E1 -1414.481,E2 -1414.481} C_VEL
LIN {X 0,Y 587.312,Z 611.45,A -85,B 0,C 180,E1 -1417.134,E2 -1417.134} C_VEL
LIN {X 0,Y 587.326,Z 611.45,A -85,B 0,C 180,E1 -1419.695,E2 -1419.695} C_VEL
LIN {X 0,Y 587.304,Z 611.449,A -85,B 0,C 180,E1 -1421.872,E2 -1421.872} C_VEL
LIN {X 0,Y 587.315,Z 611.447,A -85,B 0,C 180,E1 -1424.024,E2 -1424.024} C_VEL
LIN {X 0,Y 587.356,Z 611.442,A -85,B 0,C 180,E1 -1426.154,E2 -1426.154} C_VEL
LIN {X 0,Y 587.341,Z 611.442,A -85,B 0,C 180,E1 -1428.962,E2 -1428.962} C_VEL
LIN {X 0,Y 587.365,Z 611.448,A -85,B 0,C 180,E1 -1431.744,E2 -1431.744} C_VEL
LIN {X 0,Y 587.347,Z 611.441,A -85,B 0,C 180,E1 -1434.507,E2 -1434.507} C_VEL
LIN {X 0,Y 587.362,Z 611.442,A -85,B 0,C 180,E1 -1437.256,E2 -1437.256} C_VEL
LIN {X 0,Y 587.389,Z 611.442,A -85,B 0,C 180,E1 -1440,E2 -1440} C_VEL
LIN {X 0,Y 587.376,Z 611.437,A -85,B 0,C 180,E1 -1442.743,E2 -1442.743} C_VEL
LIN {X 0,Y 587.35,Z 611.445,A -85,B 0,C 180,E1 -1445.493,E2 -1445.493} C_VEL
LIN {X 0,Y 587.368,Z 611.444,A -85,B 0,C 180,E1 -1448.255,E2 -1448.255} C_VEL
LIN {X 0,Y 587.352,Z 611.44,A -85,B 0,C 180,E1 -1451.133,E2 -1451.133} C_VEL
LIN {X 0,Y 587.368,Z 611.445,A -85,B 0,C 180,E1 -1454.26,E2 -1454.26} C_VEL
LIN {X 0,Y 587.351,Z 611.441,A -85,B 0,C 180,E1 -1457.406,E2 -1457.406} C_VEL
LIN {X 0,Y 587.334,Z 611.45,A -85,B 0,C 180,E1 -1460.305,E2 -1460.305} C_VEL
LIN {X 0,Y 587.317,Z 611.444,A -85,B 0,C 180,E1 -1463.259,E2 -1463.259} C_VEL
LIN {X 0,Y 587.333,Z 611.444,A -85,B 0,C 180,E1 -1465.517,E2 -1465.517} C_VEL
LIN {X 0,Y 587.35,Z 611.444,A -85,B 0,C 180,E1 -1467.818,E2 -1467.818} C_VEL
LIN {X 0,Y 587.341,Z 611.449,A -85,B 0,C 180,E1 -1470.51,E2 -1470.51} C_VEL
LIN {X 0,Y 587.338,Z 611.442,A -85,B 0,C 180,E1 -1473.396,E2 -1473.396} C_VEL
LIN {X 0,Y 587.297,Z 611.45,A -85,B 0,C 180,E1 -1475.9,E2 -1475.9} C_VEL
LIN {X 0,Y 587.335,Z 611.453,A -85,B 0,C 180,E1 -1478.479,E2 -1478.479} C_VEL
LIN {X 0,Y 587.339,Z 611.443,A -85,B 0,C 180,E1 -1481.157,E2 -1481.157} C_VEL
LIN {X 0,Y 587.329,Z 611.447,A -85,B 0,C 180,E1 -1484.113,E2 -1484.113} C_VEL
LIN {X 0,Y 587.317,Z 611.448,A -85,B 0,C 180,E1 -1486.994,E2 -1486.994} C_VEL
LIN {X 0,Y 587.318,Z 611.445,A -85,B 0,C 180,E1 -1489.746,E2 -1489.746} C_VEL
LIN {X 0,Y 587.347,Z 611.447,A -85,B 0,C 180,E1 -1492.392,E2 -1492.392} C_VEL
LIN {X 0,Y 587.353,Z 611.447,A -85,B 0,C 180,E1 -1494.946,E2 -1494.946} C_VEL
LIN {X 0,Y 587.342,Z 611.443,A -85,B 0,C 180,E1 -1497.421,E2 -1497.421} C_VEL
LIN {X 0,Y 587.338,Z 611.443,A -85,B 0,C 180,E1 -1499.83,E2 -1499.83} C_VEL
LIN {X 0,Y 587.354,Z 611.444,A -85,B 0,C 180,E1 -1502.307,E2 -1502.307} C_VEL
LIN {X 0,Y 587.341,Z 611.448,A -85,B 0,C 180,E1 -1504.484,E2 -1504.484} C_VEL
LIN {X 0,Y 587.367,Z 611.587,A -85,B 0,C 180,E1 -1505.417,E2 -1505.417} C_VEL
LIN {X 0,Y 588.079,Z 616.024,A -85,B 0,C 180,E1 -1506.026,E2 -1506.026} C_VEL
LIN {X 0,Y 587.873,Z 637.906,A -85,B 0,C 180,E1 -1508.826,E2 -1508.826} C_VEL
LIN {X 0,Y 587.7,Z 660.81,A -85,B 0,C 180,E1 -1511.705,E2 -1511.705} C_VEL
LIN {X 0,Y 587.602,Z 676.431,A -85,B 0,C 180,E1 -1513.642,E2 -1513.642} C_VEL
LIN {X 0,Y 588.193,Z 680.605,A -85,B 0,C 180,E1 -1513.715,E2 -1513.715} C_VEL
LIN {X 0,Y 587.99,Z 814.879,A -85,B 0,C 180,E1 -1515.397,E2 -1515.397} C_VEL
LIN {X 0,Y 587.903,Z 829.29,A -85,B 0,C 180,E1 -1515.723,E2 -1515.723} C_VEL
LIN {X 0,Y 587.822,Z 843.833,A -85,B 0,C 180,E1 -1516.209,E2 -1516.209} C_VEL
LIN {X 0,Y 587.727,Z 856.634,A -85,B 0,C 180,E1 -1516.78,E2 -1516.78} C_VEL
LIN {X 0,Y 587.63,Z 869.094,A -85,B 0,C 180,E1 -1517.48,E2 -1517.48} C_VEL
LIN {X 0,Y 587.513,Z 880.473,A -85,B 0,C 180,E1 -1518.266,E2 -1518.266} C_VEL
LIN {X 0,Y 587.467,Z 890.932,A -85,B 0,C 180,E1 -1519.139,E2 -1519.139} C_VEL
LIN {X 0,Y 587.353,Z 901.333,A -85,B 0,C 180,E1 -1520.182,E2 -1520.182} C_VEL
LIN {X 0,Y 587.311,Z 909.912,A -85,B 0,C 180,E1 -1521.224,E2 -1521.224} C_VEL
LIN {X 0,Y 587.249,Z 918.114,A -85,B 0,C 180,E1 -1522.435,E2 -1522.435} C_VEL
LIN {X 0,Y 587.179,Z 924.681,A -85,B 0,C 180,E1 -1523.635,E2 -1523.635} C_VEL
LIN {X 0,Y 587.158,Z 929.961,A -85,B 0,C 180,E1 -1524.849,E2 -1524.849} C_VEL
LIN {X 0,Y 587.18,Z 933.442,A -85,B 0,C 180,E1 -1525.882,E2 -1525.882} C_VEL
LIN {X 0,Y 587.13,Z 936.831,A -85,B 0,C 180,E1 -1527.256,E2 -1527.256} C_VEL
LIN {X 0,Y 587.141,Z 938.831,A -85,B 0,C 180,E1 -1528.628,E2 -1528.628} C_VEL
LIN {X 0,Y 587.135,Z 939.5,A -85,B 0,C 180,E1 -1530,E2 -1530} C_VEL
LIN {X 0,Y 587.141,Z 938.832,A -85,B 0,C 180,E1 -1531.372,E2 -1531.372} C_VEL
LIN {X 0,Y 587.13,Z 936.832,A -85,B 0,C 180,E1 -1532.744,E2 -1532.744} C_VEL
LIN {X 0,Y 587.18,Z 933.443,A -85,B 0,C 180,E1 -1534.118,E2 -1534.118} C_VEL
LIN {X 0,Y 587.199,Z 928.568,A -85,B 0,C 180,E1 -1535.494,E2 -1535.494} C_VEL
LIN {X 0,Y 587.209,Z 922.052,A -85,B 0,C 180,E1 -1536.874,E2 -1536.874} C_VEL
LIN {X 0,Y 587.268,Z 914.799,A -85,B 0,C 180,E1 -1538.083,E2 -1538.083} C_VEL
LIN {X 0,Y 587.322,Z 905.823,A -85,B 0,C 180,E1 -1539.296,E2 -1539.296} C_VEL
LIN {X 0,Y 587.372,Z 896.391,A -85,B 0,C 180,E1 -1540.339,E2 -1540.339} C_VEL
LIN {X 0,Y 587.475,Z 886.025,A -85,B 0,C 180,E1 -1541.29,E2 -1541.29} C_VEL
LIN {X 0,Y 587.571,Z 874.429,A -85,B 0,C 180,E1 -1542.17,E2 -1542.17} C_VEL
LIN {X 0,Y 587.665,Z 861.647,A -85,B 0,C 180,E1 -1542.958,E2 -1542.958} C_VEL
LIN {X 0,Y 587.813,Z 849.161,A -85,B 0,C 180,E1 -1543.57,E2 -1543.57} C_VEL
LIN {X 0,Y 587.896,Z 835.73,A -85,B 0,C 180,E1 -1544.081,E2 -1544.081} C_VEL
LIN {X 0,Y 587.962,Z 821.304,A -85,B 0,C 180,E1 -1544.477,E2 -1544.477} C_VEL
LIN {X 0,Y 588.01,Z 807.603,A -85,B 0,C 180,E1 -1544.713,E2 -1544.713} C_VEL
LIN {X 0,Y 588.071,Z 679.163,A -85,B 0,C 180,E1 -1546.307,E2 -1546.307} C_VEL
LIN {X 0,Y 587.594,Z 676.342,A -85,B 0,C 180,E1 -1546.369,E2 -1546.369} C_VEL
LIN {X 0,Y 587.722,Z 654.008,A -85,B 0,C 180,E1 -1549.146,E2 -1549.146} C_VEL
LIN {X 0,Y 587.917,Z 633.362,A -85,B 0,C 180,E1 -1551.751,E2 -1551.751} C_VEL
LIN {X 0,Y 588.05,Z 614.748,A -85,B 0,C 180,E1 -1554.141,E2 -1554.141} C_VEL
LIN {X 0,Y 587.334,Z 611.452,A -85,B 0,C 180,E1 -1554.632,E2 -1554.632} C_VEL
LIN {X 0,Y 587.332,Z 611.453,A -85,B 0,C 180,E1 -1557.046,E2 -1557.046} C_VEL
LIN {X 0,Y 587.35,Z 611.449,A -85,B 0,C 180,E1 -1559.379,E2 -1559.379} C_VEL
LIN {X 0,Y 587.356,Z 611.442,A -85,B 0,C 180,E1 -1561.837,E2 -1561.837} C_VEL
LIN {X 0,Y 587.358,Z 611.439,A -85,B 0,C 180,E1 -1564.349,E2 -1564.349} C_VEL
LIN {X 0,Y 587.354,Z 611.442,A -85,B 0,C 180,E1 -1566.747,E2 -1566.747} C_VEL
LIN {X 0,Y 587.347,Z 611.452,A -85,B 0,C 180,E1 -1569.359,E2 -1569.359} C_VEL
LIN {X 0,Y 587.336,Z 611.444,A -85,B 0,C 180,E1 -1572.108,E2 -1572.108} C_VEL
LIN {X 0,Y 587.317,Z 611.448,A -85,B 0,C 180,E1 -1575.089,E2 -1575.089} C_VEL
LIN {X 0,Y 587.355,Z 611.444,A -85,B 0,C 180,E1 -1577.928,E2 -1577.928} C_VEL
LIN {X 0,Y 587.336,Z 611.445,A -85,B 0,C 180,E1 -1581.058,E2 -1581.058} C_VEL
LIN {X 0,Y 587.356,Z 611.443,A -85,B 0,C 180,E1 -1583.292,E2 -1583.292} C_VEL
LIN {X 0,Y 587.37,Z 611.447,A -85,B 0,C 180,E1 -1585.781,E2 -1585.781} C_VEL
LIN {X 0,Y 587.356,Z 611.44,A -85,B 0,C 180,E1 -1588.232,E2 -1588.232} C_VEL
LIN {X 0,Y 587.352,Z 611.44,A -85,B 0,C 180,E1 -1590.866,E2 -1590.866} C_VEL
LIN {X 0,Y 587.36,Z 611.45,A -85,B 0,C 180,E1 -1593.819,E2 -1593.819} C_VEL
LIN {X 0,Y 587.34,Z 611.451,A -85,B 0,C 180,E1 -1595.994,E2 -1595.994} C_VEL
LIN {X 0,Y 587.325,Z 611.449,A -85,B 0,C 180,E1 -1598.226,E2 -1598.226} C_VEL
LIN {X 0,Y 587.353,Z 611.44,A -85,B 0,C 180,E1 -1601.151,E2 -1601.151} C_VEL
LIN {X 0,Y 587.356,Z 611.441,A -85,B 0,C 180,E1 -1603.311,E2 -1603.311} C_VEL
LIN {X 0,Y 587.361,Z 611.449,A -85,B 0,C 180,E1 -1606.154,E2 -1606.154} C_VEL
LIN {X 0,Y 587.345,Z 611.441,A -85,B 0,C 180,E1 -1608.963,E2 -1608.963} C_VEL
LIN {X 0,Y 587.368,Z 611.441,A -85,B 0,C 180,E1 -1611.745,E2 -1611.745} C_VEL
LIN {X 0,Y 587.351,Z 611.446,A -85,B 0,C 180,E1 -1614.507,E2 -1614.507} C_VEL
LIN {X 0,Y 587.378,Z 611.437,A -85,B 0,C 180,E1 -1617.257,E2 -1617.257} C_VEL
LIN {X 0,Y 587.385,Z 611.441,A -85,B 0,C 180,E1 -1620,E2 -1620} C_VEL
LIN {X 0,Y 587.369,Z 611.443,A -85,B 0,C 180,E1 -1622.743,E2 -1622.743} C_VEL
LIN {X 0,Y 587.356,Z 611.439,A -85,B 0,C 180,E1 -1625.493,E2 -1625.493} C_VEL
LIN {X 0,Y 587.369,Z 611.445,A -85,B 0,C 180,E1 -1628.255,E2 -1628.255} C_VEL
LIN {X 0,Y 587.351,Z 611.442,A -85,B 0,C 180,E1 -1631.134,E2 -1631.134} C_VEL
LIN {X 0,Y 587.368,Z 611.443,A -85,B 0,C 180,E1 -1634.26,E2 -1634.26} C_VEL
LIN {X 0,Y 587.348,Z 611.442,A -85,B 0,C 180,E1 -1637.406,E2 -1637.406} C_VEL
LIN {X 0,Y 587.309,Z 611.448,A -85,B 0,C 180,E1 -1638.311,E2 -1638.311} C_VEL
LIN {X 0,Y 586.668,Z 611.534,A -85,B 0,C 180,E1 -1638.883,E2 -1638.883} C_VEL
LIN {X 0,Y 583.845,Z 611.885,A -85,B 0,C 180,E1 -1639.812,E2 -1639.812} C_VEL
LIN {X 0,Y 581.435,Z 612.185,A -85,B 0,C 180,E1 -1640.559,E2 -1640.559} C_VEL
LIN {X 0,Y 580.381,Z 612.313,A -85,B 0,C 180,E1 -1641.135,E2 -1641.135} C_VEL
LIN {X 0,Y 580.285,Z 612.323,A -85,B 0,C 180,E1 -1641.33,E2 -1641.33} C_VEL
LIN {X 0,Y 580.298,Z 612.321,A -85,B 0,C 180,E1 -1644.317,E2 -1644.317} C_VEL
LIN {X 0,Y 580.268,Z 612.33,A -85,B 0,C 180,E1 -1646.624,E2 -1646.624} C_VEL
LIN {X 0,Y 580.297,Z 612.321,A -85,B 0,C 180,E1 -1649.309,E2 -1649.309} C_VEL
LIN {X 0,Y 580.3,Z 612.32,A -85,B 0,C 180,E1 -1652.201,E2 -1652.201} C_VEL
LIN {X 0,Y 580.287,Z 612.326,A -85,B 0,C 180,E1 -1654.697,E2 -1654.697} C_VEL
LIN {X 0,Y 580.298,Z 612.326,A -85,B 0,C 180,E1 -1657.269,E2 -1657.269} C_VEL
LIN {X 0,Y 580.287,Z 612.32,A -85,B 0,C 180,E1 -1660.27,E2 -1660.27} C_VEL
LIN {X 0,Y 580.26,Z 612.328,A -85,B 0,C 180,E1 -1662.708,E2 -1662.708} C_VEL
LIN {X 0,Y 580.253,Z 612.329,A -85,B 0,C 180,E1 -1665.611,E2 -1665.611} C_VEL
LIN {X 0,Y 580.272,Z 612.325,A -85,B 0,C 180,E1 -1668.67,E2 -1668.67} C_VEL
LIN {X 0,Y 580.267,Z 612.329,A -85,B 0,C 180,E1 -1670.964,E2 -1670.964} C_VEL
LIN {X 0,Y 580.266,Z 612.329,A -85,B 0,C 180,E1 -1673.596,E2 -1673.596} C_VEL
LIN {X 0,Y 580.278,Z 612.322,A -85,B 0,C 180,E1 -1676.143,E2 -1676.143} C_VEL
LIN {X 0,Y 580.265,Z 612.324,A -85,B 0,C 180,E1 -1678.614,E2 -1678.614} C_VEL
LIN {X 0,Y 580.285,Z 612.325,A -85,B 0,C 180,E1 -1681.023,E2 -1681.023} C_VEL
LIN {X 0,Y 580.269,Z 612.329,A -85,B 0,C 180,E1 -1684.246,E2 -1684.246} C_VEL
LIN {X 0,Y 580.284,Z 612.38,A -85,B 0,C 180,E1 -1684.343,E2 -1684.343} C_VEL
LIN {X 0,Y 580.669,Z 617.695,A -85,B 0,C 180,E1 -1685.197,E2 -1685.197} C_VEL
LIN {X 0,Y 580.517,Z 636.488,A -85,B 0,C 180,E1 -1688.125,E2 -1688.125} C_VEL
LIN {X 0,Y 580.502,Z 638.909,A -85,B 0,C 180,E1 -1688.499,E2 -1688.499} C_VEL
LIN {X 0,Y 581.404,Z 644.774,A -85,B 0,C 180,E1 -1688.604,E2 -1688.604} C_VEL
LIN {X 0,Y 581.101,Z 775.687,A -85,B 0,C 180,E1 -1690.261,E2 -1690.261} C_VEL
LIN {X 0,Y 581.033,Z 790.356,A -85,B 0,C 180,E1 -1690.598,E2 -1690.598} C_VEL
LIN {X 0,Y 580.925,Z 804.451,A -85,B 0,C 180,E1 -1691.072,E2 -1691.072} C_VEL
LIN {X 0,Y 580.754,Z 817.599,A -85,B 0,C 180,E1 -1691.661,E2 -1691.661} C_VEL
LIN {X 0,Y 580.651,Z 830.324,A -85,B 0,C 180,E1 -1692.387,E2 -1692.387} C_VEL
LIN {X 0,Y 580.535,Z 841.889,A -85,B 0,C 180,E1 -1693.2,E2 -1693.2} C_VEL
LIN {X 0,Y 580.426,Z 853.456,A -85,B 0,C 180,E1 -1694.191,E2 -1694.191} C_VEL
LIN {X 0,Y 580.312,Z 863.708,A -85,B 0,C 180,E1 -1695.266,E2 -1695.266} C_VEL
LIN {X 0,Y 580.227,Z 872.181,A -85,B 0,C 180,E1 -1696.338,E2 -1696.338} C_VEL
LIN {X 0,Y 580.154,Z 880.246,A -85,B 0,C 180,E1 -1697.583,E2 -1697.583} C_VEL
LIN {X 0,Y 580.081,Z 887.16,A -85,B 0,C 180,E1 -1698.922,E2 -1698.922} C_VEL
LIN {X 0,Y 580.084,Z 892.393,A -85,B 0,C 180,E1 -1700.234,E2 -1700.234} C_VEL
LIN {X 0,Y 580.068,Z 896.491,A -85,B 0,C 180,E1 -1701.64,E2 -1701.64} C_VEL
LIN {X 0,Y 580.062,Z 899.124,A -85,B 0,C 180,E1 -1703.041,E2 -1703.041} C_VEL
LIN {X 0,Y 580.088,Z 900.369,A -85,B 0,C 180,E1 -1704.438,E2 -1704.438} C_VEL
LIN {X 0,Y 580.084,Z 900.271,A -85,B 0,C 180,E1 -1705.831,E2 -1705.831} C_VEL
LIN {X 0,Y 580.036,Z 898.851,A -85,B 0,C 180,E1 -1707.222,E2 -1707.222} C_VEL
LIN {X 0,Y 580.048,Z 896.078,A -85,B 0,C 180,E1 -1708.612,E2 -1708.612} C_VEL
LIN {X 0,Y 580.07,Z 891.88,A -85,B 0,C 180,E1 -1710,E2 -1710} C_VEL
LIN {X 0,Y 580.083,Z 886.141,A -85,B 0,C 180,E1 -1711.389,E2 -1711.389} C_VEL
LIN {X 0,Y 580.209,Z 879.683,A -85,B 0,C 180,E1 -1712.604,E2 -1712.604} C_VEL
LIN {X 0,Y 580.26,Z 871.7,A -85,B 0,C 180,E1 -1713.82,E2 -1713.82} C_VEL
LIN {X 0,Y 580.352,Z 863.37,A -85,B 0,C 180,E1 -1714.863,E2 -1714.863} C_VEL
LIN {X 0,Y 580.421,Z 853.371,A -85,B 0,C 180,E1 -1715.908,E2 -1715.908} C_VEL
LIN {X 0,Y 580.517,Z 842.938,A -85,B 0,C 180,E1 -1716.81,E2 -1716.81} C_VEL
LIN {X 0,Y 580.656,Z 831.151,A -85,B 0,C 180,E1 -1717.651,E2 -1717.651} C_VEL
LIN {X 0,Y 580.782,Z 819.144,A -85,B 0,C 180,E1 -1718.35,E2 -1718.35} C_VEL
LIN {X 0,Y 580.943,Z 806.978,A -85,B 0,C 180,E1 -1718.917,E2 -1718.917} C_VEL
LIN {X 0,Y 581.027,Z 793.556,A -85,B 0,C 180,E1 -1719.398,E2 -1719.398} C_VEL
LIN {X 0,Y 581.09,Z 779.81,A -85,B 0,C 180,E1 -1719.749,E2 -1719.749} C_VEL
LIN {X 0,Y 581.116,Z 762.63,A -85,B 0,C 180,E1 -1720.012,E2 -1720.012} C_VEL
LIN {X 0,Y 581.295,Z 643.255,A -85,B 0,C 180,E1 -1721.508,E2 -1721.508} C_VEL
LIN {X 0,Y 580.473,Z 638.93,A -85,B 0,C 180,E1 -1721.588,E2 -1721.588} C_VEL
LIN {X 0,Y 580.629,Z 621.394,A -85,B 0,C 180,E1 -1724.313,E2 -1724.313} C_VEL
LIN {X 0,Y 580.588,Z 614.217,A -85,B 0,C 180,E1 -1725.445,E2 -1725.445} C_VEL
LIN {X 0,Y 580.275,Z 612.329,A -85,B 0,C 180,E1 -1725.769,E2 -1725.769} C_VEL
LIN {X 0,Y 580.237,Z 612.335,A -85,B 0,C 180,E1 -1728.356,E2 -1728.356} C_VEL
LIN {X 0,Y 580.306,Z 612.322,A -85,B 0,C 180,E1 -1731.165,E2 -1731.165} C_VEL
LIN {X 0,Y 580.251,Z 612.326,A -85,B 0,C 180,E1 -1733.559,E2 -1733.559} C_VEL
LIN {X 0,Y 580.233,Z 612.337,A -85,B 0,C 180,E1 -1736.626,E2 -1736.626} C_VEL
LIN {X 0,Y 580.264,Z 612.326,A -85,B 0,C 180,E1 -1739.302,E2 -1739.302} C_VEL
LIN {X 0,Y 580.281,Z 612.323,A -85,B 0,C 180,E1 -1742.202,E2 -1742.202} C_VEL
LIN {X 0,Y 580.274,Z 612.33,A -85,B 0,C 180,E1 -1744.698,E2 -1744.698} C_VEL
LIN {X 0,Y 580.272,Z 612.327,A -85,B 0,C 180,E1 -1747.271,E2 -1747.271} C_VEL
LIN {X 0,Y 580.275,Z 612.321,A -85,B 0,C 180,E1 -1750.268,E2 -1750.268} C_VEL
LIN {X 0,Y 580.236,Z 612.331,A -85,B 0,C 180,E1 -1753.386,E2 -1753.386} C_VEL
LIN {X 0,Y 580.253,Z 612.327,A -85,B 0,C 180,E1 -1755.611,E2 -1755.611} C_VEL
LIN {X 0,Y 580.239,Z 612.327,A -85,B 0,C 180,E1 -1758.227,E2 -1758.227} C_VEL
LIN {X 0,Y 580.263,Z 612.331,A -85,B 0,C 180,E1 -1760.963,E2 -1760.963} C_VEL
LIN {X 0,Y 580.245,Z 612.328,A -85,B 0,C 180,E1 -1763.594,E2 -1763.594} C_VEL
LIN {X 0,Y 580.279,Z 612.321,A -85,B 0,C 180,E1 -1766.142,E2 -1766.142} C_VEL
LIN {X 0,Y 580.268,Z 612.324,A -85,B 0,C 180,E1 -1768.614,E2 -1768.614} C_VEL
LIN {X 0,Y 580.288,Z 612.325,A -85,B 0,C 180,E1 -1771.023,E2 -1771.023} C_VEL
LIN {X 0,Y 580.247,Z 612.326,A -85,B 0,C 180,E1 -1774.148,E2 -1774.148} C_VEL
LIN {X 0,Y 580.267,Z 612.322,A -85,B 0,C 180,E1 -1776.441,E2 -1776.441} C_VEL
LIN {X 0,Y 580.274,Z 612.333,A -85,B 0,C 180,E1 -1779.437,E2 -1779.437} C_VEL
LIN {X 0,Y 580.264,Z 612.329,A -85,B 0,C 180,E1 -1781.645,E2 -1781.645} C_VEL
LIN {X 0,Y 580.269,Z 612.328,A -85,B 0,C 180,E1 -1783.825,E2 -1783.825} C_VEL
LIN {X 0,Y 580.326,Z 612.319,A -85,B 0,C 180,E1 -1785.983,E2 -1785.983} C_VEL
LIN {X 0,Y 580.309,Z 612.317,A -85,B 0,C 180,E1 -1788.827,E2 -1788.827} C_VEL
LIN {X 0,Y 580.327,Z 612.326,A -85,B 0,C 180,E1 -1791.644,E2 -1791.644} C_VEL
LIN {X 0,Y 580.314,Z 612.318,A -85,B 0,C 180,E1 -1794.44,E2 -1794.44} C_VEL
LIN {X 0,Y 580.33,Z 612.317,A -85,B 0,C 180,E1 -1797.223,E2 -1797.223} C_VEL
LIN {X 0,Y 580.358,Z 612.318,A -85,B 0,C 180,E1 -1800,E2 -1800} C_VEL
LIN {X 0,Y 580.342,Z 612.314,A -85,B 0,C 180,E1 -1802.776,E2 -1802.776} C_VEL
LIN {X 0,Y 580.318,Z 612.321,A -85,B 0,C 180,E1 -1805.56,E2 -1805.56} C_VEL
LIN {X 0,Y 580.331,Z 612.319,A -85,B 0,C 180,E1 -1808.356,E2 -1808.356} C_VEL
LIN {X 0,Y 580.304,Z 612.318,A -85,B 0,C 180,E1 -1811.191,E2 -1811.191} C_VEL
LIN {X 0,Y 580.328,Z 612.326,A -85,B 0,C 180,E1 -1814.017,E2 -1814.017} C_VEL
LIN {X 0,Y 580.316,Z 612.317,A -85,B 0,C 180,E1 -1816.914,E2 -1816.914} C_VEL
LIN {X 0,Y 580.308,Z 612.323,A -85,B 0,C 180,E1 -1819.822,E2 -1819.822} C_VEL
LIN {X 0,Y 580.294,Z 612.321,A -85,B 0,C 180,E1 -1822.802,E2 -1822.802} C_VEL
LIN {X 0,Y 580.308,Z 612.318,A -85,B 0,C 180,E1 -1825.08,E2 -1825.08} C_VEL
LIN {X 0,Y 580.303,Z 612.327,A -85,B 0,C 180,E1 -1828.185,E2 -1828.185} C_VEL
LIN {X 0,Y 580.29,Z 612.324,A -85,B 0,C 180,E1 -1830.695,E2 -1830.695} C_VEL
LIN {X 0,Y 580.307,Z 612.318,A -85,B 0,C 180,E1 -1833.316,E2 -1833.316} C_VEL
LIN {X 0,Y 580.253,Z 612.326,A -85,B 0,C 180,E1 -1835.757,E2 -1835.757} C_VEL
LIN {X 0,Y 580.291,Z 612.326,A -85,B 0,C 180,E1 -1838.146,E2 -1838.146} C_VEL
LIN {X 0,Y 580.302,Z 612.323,A -85,B 0,C 180,E1 -1840.843,E2 -1840.843} C_VEL
LIN {X 0,Y 580.281,Z 612.321,A -85,B 0,C 180,E1 -1843.658,E2 -1843.658} C_VEL
LIN {X 0,Y 580.279,Z 612.331,A -85,B 0,C 180,E1 -1846.609,E2 -1846.609} C_VEL
LIN {X 0,Y 580.303,Z 612.321,A -85,B 0,C 180,E1 -1849.157,E2 -1849.157} C_VEL
LIN {X 0,Y 580.292,Z 612.321,A -85,B 0,C 180,E1 -1851.927,E2 -1851.927} C_VEL
LIN {X 0,Y 580.309,Z 612.325,A -85,B 0,C 180,E1 -1854.457,E2 -1854.457} C_VEL
LIN {X 0,Y 580.294,Z 612.327,A -85,B 0,C 180,E1 -1856.975,E2 -1856.975} C_VEL
LIN {X 0,Y 580.304,Z 612.321,A -85,B 0,C 180,E1 -1859.425,E2 -1859.425} C_VEL
LIN {X 0,Y 580.3,Z 612.321,A -85,B 0,C 180,E1 -1862.141,E2 -1862.141} C_VEL
LIN {X 0,Y 580.311,Z 612.327,A -85,B 0,C 180,E1 -1864.92,E2 -1864.92} C_VEL
LIN {X 0,Y 580.34,Z 612.479,A -85,B 0,C 180,E1 -1865.217,E2 -1865.217} C_VEL
LIN {X 0,Y 581.242,Z 617.469,A -85,B 0,C 180,E1 -1865.915,E2 -1865.915} C_VEL
LIN {X 0,Y 580.965,Z 639.14,A -85,B 0,C 180,E1 -1868.721,E2 -1868.721} C_VEL
LIN {X 0,Y 580.768,Z 660.81,A -85,B 0,C 180,E1 -1871.479,E2 -1871.479} C_VEL
LIN {X 0,Y 580.636,Z 676.431,A -85,B 0,C 180,E1 -1873.44,E2 -1873.44} C_VEL
LIN {X 0,Y 581.404,Z 682.394,A -85,B 0,C 180,E1 -1873.542,E2 -1873.542} C_VEL
LIN {X 0,Y 581.117,Z 814.879,A -85,B 0,C 180,E1 -1875.22,E2 -1875.22} C_VEL
LIN {X 0,Y 581.022,Z 829.46,A -85,B 0,C 180,E1 -1875.556,E2 -1875.556} C_VEL
LIN {X 0,Y 580.924,Z 843.834,A -85,B 0,C 180,E1 -1876.042,E2 -1876.042} C_VEL
LIN {X 0,Y 580.798,Z 856.636,A -85,B 0,C 180,E1 -1876.619,E2 -1876.619} C_VEL
LIN {X 0,Y 580.661,Z 869.095,A -85,B 0,C 180,E1 -1877.328,E2 -1877.328} C_VEL
LIN {X 0,Y 580.525,Z 881.637,A -85,B 0,C 180,E1 -1878.212,E2 -1878.212} C_VEL
LIN {X 0,Y 580.441,Z 892.906,A -85,B 0,C 180,E1 -1879.19,E2 -1879.19} C_VEL
LIN {X 0,Y 580.275,Z 902.85,A -85,B 0,C 180,E1 -1880.238,E2 -1880.238} C_VEL
LIN {X 0,Y 580.241,Z 911.17,A -85,B 0,C 180,E1 -1881.292,E2 -1881.292} C_VEL
LIN {X 0,Y 580.166,Z 919.125,A -85,B 0,C 180,E1 -1882.517,E2 -1882.517} C_VEL
LIN {X 0,Y 580.102,Z 925.527,A -85,B 0,C 180,E1 -1883.74,E2 -1883.74} C_VEL
LIN {X 0,Y 580.077,Z 929.961,A -85,B 0,C 180,E1 -1884.786,E2 -1884.786} C_VEL
LIN {X 0,Y 580.103,Z 933.442,A -85,B 0,C 180,E1 -1885.831,E2 -1885.831} C_VEL
LIN {X 0,Y 580.04,Z 936.831,A -85,B 0,C 180,E1 -1887.222,E2 -1887.222} C_VEL
LIN {X 0,Y 580.041,Z 938.832,A -85,B 0,C 180,E1 -1888.611,E2 -1888.611} C_VEL
LIN {X 0,Y 580.036,Z 939.5,A -85,B 0,C 180,E1 -1890,E2 -1890} C_VEL
LIN {X 0,Y 580.041,Z 938.832,A -85,B 0,C 180,E1 -1891.389,E2 -1891.389} C_VEL
LIN {X 0,Y 580.04,Z 936.833,A -85,B 0,C 180,E1 -1892.778,E2 -1892.778} C_VEL
LIN {X 0,Y 580.103,Z 933.443,A -85,B 0,C 180,E1 -1894.168,E2 -1894.168} C_VEL
LIN {X 0,Y 580.128,Z 928.568,A -85,B 0,C 180,E1 -1895.562,E2 -1895.562} C_VEL
LIN {X 0,Y 580.141,Z 922.052,A -85,B 0,C 180,E1 -1896.958,E2 -1896.958} C_VEL
LIN {X 0,Y 580.192,Z 914.8,A -85,B 0,C 180,E1 -1898.183,E2 -1898.183} C_VEL
LIN {X 0,Y 580.284,Z 905.823,A -85,B 0,C 180,E1 -1899.41,E2 -1899.41} C_VEL
LIN {X 0,Y 580.356,Z 896.392,A -85,B 0,C 180,E1 -1900.466,E2 -1900.466} C_VEL
LIN {X 0,Y 580.475,Z 886.318,A -85,B 0,C 180,E1 -1901.404,E2 -1901.404} C_VEL
LIN {X 0,Y 580.594,Z 874.43,A -85,B 0,C 180,E1 -1902.319,E2 -1902.319} C_VEL
LIN {X 0,Y 580.724,Z 861.649,A -85,B 0,C 180,E1 -1903.115,E2 -1903.115} C_VEL
LIN {X 0,Y 580.909,Z 849.16,A -85,B 0,C 180,E1 -1903.735,E2 -1903.735} C_VEL
LIN {X 0,Y 581.001,Z 836.25,A -85,B 0,C 180,E1 -1904.234,E2 -1904.234} C_VEL
LIN {X 0,Y 581.082,Z 822.196,A -85,B 0,C 180,E1 -1904.63,E2 -1904.63} C_VEL
LIN {X 0,Y 581.149,Z 807.603,A -85,B 0,C 180,E1 -1904.891,E2 -1904.891} C_VEL
LIN {X 0,Y 581.297,Z 680.291,A -85,B 0,C 180,E1 -1906.488,E2 -1906.488} C_VEL
LIN {X 0,Y 580.643,Z 676.342,A -85,B 0,C 180,E1 -1906.571,E2 -1906.571} C_VEL
LIN {X 0,Y 580.829,Z 653.21,A -85,B 0,C 180,E1 -1909.484,E2 -1909.484} C_VEL
LIN {X 0,Y 581.097,Z 630.473,A -85,B 0,C 180,E1 -1912.394,E2 -1912.394} C_VEL
LIN {X 0,Y 581.241,Z 617.47,A -85,B 0,C 180,E1 -1914.084,E2 -1914.084} C_VEL
LIN {X 0,Y 580.327,Z 612.326,A -85,B 0,C 180,E1 -1914.81,E2 -1914.81} C_VEL
LIN {X 0,Y 580.29,Z 612.328,A -85,B 0,C 180,E1 -1917.402,E2 -1917.402} C_VEL
LIN {X 0,Y 580.291,Z 612.323,A -85,B 0,C 180,E1 -1919.773,E2 -1919.773} C_VEL
LIN {X 0,Y 580.304,Z 612.318,A -85,B 0,C 180,E1 -1922.2,E2 -1922.2} C_VEL
LIN {X 0,Y 580.303,Z 612.32,A -85,B 0,C 180,E1 -1924.695,E2 -1924.695} C_VEL
LIN {X 0,Y 580.302,Z 612.328,A -85,B 0,C 180,E1 -1927.268,E2 -1927.268} C_VEL
LIN {X 0,Y 580.301,Z 612.318,A -85,B 0,C 180,E1 -1930.272,E2 -1930.272} C_VEL
LIN {X 0,Y 580.28,Z 612.322,A -85,B 0,C 180,E1 -1932.706,E2 -1932.706} C_VEL
LIN {X 0,Y 580.271,Z 612.332,A -85,B 0,C 180,E1 -1935.609,E2 -1935.609} C_VEL
LIN {X 0,Y 580.316,Z 612.317,A -85,B 0,C 180,E1 -1938.234,E2 -1938.234} C_VEL
LIN {X 0,Y 580.291,Z 612.321,A -85,B 0,C 180,E1 -1940.966,E2 -1940.966} C_VEL
LIN {X 0,Y 580.299,Z 612.327,A -85,B 0,C 180,E1 -1943.599,E2 -1943.599} C_VEL
LIN {X 0,Y 580.322,Z 612.319,A -85,B 0,C 180,E1 -1946.146,E2 -1946.146} C_VEL
LIN {X 0,Y 580.291,Z 612.317,A -85,B 0,C 180,E1 -1948.615,E2 -1948.615} C_VEL
LIN {X 0,Y 580.296,Z 612.319,A -85,B 0,C 180,E1 -1951.024,E2 -1951.024} C_VEL
LIN {X 0,Y 580.293,Z 612.327,A -85,B 0,C 180,E1 -1953.666,E2 -1953.666} C_VEL
LIN {X 0,Y 580.304,Z 612.325,A -85,B 0,C 180,E1 -1955.684,E2 -1955.684} C_VEL
LIN {X 0,Y 580.276,Z 612.332,A -85,B 0,C 180,E1 -1957.948,E2 -1957.948} C_VEL
LIN {X 0,Y 580.321,Z 612.316,A -85,B 0,C 180,E1 -1960.914,E2 -1960.914} C_VEL
LIN {X 0,Y 580.283,Z 612.328,A -85,B 0,C 180,E1 -1963.826,E2 -1963.826} C_VEL
LIN {X 0,Y 580.328,Z 612.325,A -85,B 0,C 180,E1 -1965.983,E2 -1965.983} C_VEL
LIN {X 0,Y 580.307,Z 612.319,A -85,B 0,C 180,E1 -1968.827,E2 -1968.827} C_VEL
LIN {X 0,Y 580.331,Z 612.316,A -85,B 0,C 180,E1 -1971.644,E2 -1971.644} C_VEL
LIN {X 0,Y 580.319,Z 612.323,A -85,B 0,C 180,E1 -1974.44,E2 -1974.44} C_VEL
LIN {X 0,Y 580.343,Z 612.313,A -85,B 0,C 180,E1 -1977.224,E2 -1977.224} C_VEL
LIN {X 0,Y 580.354,Z 612.317,A -85,B 0,C 180,E1 -1980,E2 -1980} C_VEL
LIN {X 0,Y 580.336,Z 612.319,A -85,B 0,C 180,E1 -1982.777,E2 -1982.777} C_VEL
LIN {X 0,Y 580.325,Z 612.315,A -85,B 0,C 180,E1 -1985.56,E2 -1985.56} C_VEL
LIN {X 0,Y 580.331,Z 612.324,A -85,B 0,C 180,E1 -1988.356,E2 -1988.356} C_VEL
LIN {X 0,Y 580.303,Z 612.32,A -85,B 0,C 180,E1 -1991.191,E2 -1991.191} C_VEL
LIN {X 0,Y 580.326,Z 612.318,A -85,B 0,C 180,E1 -1994.017,E2 -1994.017} C_VEL
LIN {X 0,Y 580.316,Z 612.323,A -85,B 0,C 180,E1 -1996.914,E2 -1996.914} C_VEL
LIN {X 0,Y 580.288,Z 612.32,A -85,B 0,C 180,E1 -1999.823,E2 -1999.823} C_VEL
LIN {X 0,Y 580.285,Z 612.323,A -85,B 0,C 180,E1 -2001.33,E2 -2001.33} C_VEL
LIN {X 0,Y 579.585,Z 612.41,A -85,B 0,C 180,E1 -2001.909,E2 -2001.909} C_VEL
LIN {X 0,Y 576.706,Z 612.775,A -85,B 0,C 180,E1 -2002.849,E2 -2002.849} C_VEL
LIN {X 0,Y 574.312,Z 613.068,A -85,B 0,C 180,E1 -2003.605,E2 -2003.605} C_VEL
LIN {X 0,Y 573.314,Z 613.19,A -85,B 0,C 180,E1 -2004.189,E2 -2004.189} C_VEL
LIN {X 0,Y 573.248,Z 613.2,A -85,B 0,C 180,E1 -2004.387,E2 -2004.387} C_VEL
LIN {X 0,Y 573.205,Z 613.209,A -85,B 0,C 180,E1 -2006.979,E2 -2006.979} C_VEL
LIN {X 0,Y 573.241,Z 613.198,A -85,B 0,C 180,E1 -2009.487,E2 -2009.487} C_VEL
LIN {X 0,Y 573.255,Z 613.202,A -85,B 0,C 180,E1 -2012.645,E2 -2012.645} C_VEL
LIN {X 0,Y 573.206,Z 613.21,A -85,B 0,C 180,E1 -2015.188,E2 -2015.188} C_VEL
LIN {X 0,Y 573.233,Z 613.2,A -85,B 0,C 180,E1 -2017.808,E2 -2017.808} C_VEL
LIN {X 0,Y 573.248,Z 613.198,A -85,B 0,C 180,E1 -2020.525,E2 -2020.525} C_VEL
LIN {X 0,Y 573.21,Z 613.205,A -85,B 0,C 180,E1 -2023.665,E2 -2023.665} C_VEL
LIN {X 0,Y 573.205,Z 613.205,A -85,B 0,C 180,E1 -2026.638,E2 -2026.638} C_VEL
LIN {X 0,Y 573.248,Z 613.205,A -85,B 0,C 180,E1 -2029.475,E2 -2029.475} C_VEL
LIN {X 0,Y 573.231,Z 613.2,A -85,B 0,C 180,E1 -2032.192,E2 -2032.192} C_VEL
LIN {X 0,Y 573.229,Z 613.208,A -85,B 0,C 180,E1 -2035.23,E2 -2035.23} C_VEL
LIN {X 0,Y 573.242,Z 613.204,A -85,B 0,C 180,E1 -2037.774,E2 -2037.774} C_VEL
LIN {X 0,Y 573.24,Z 613.2,A -85,B 0,C 180,E1 -2040.633,E2 -2040.633} C_VEL
LIN {X 0,Y 573.196,Z 613.215,A -85,B 0,C 180,E1 -2043.517,E2 -2043.517} C_VEL
LIN {X 0,Y 573.262,Z 613.298,A -85,B 0,C 180,E1 -2044.225,E2 -2044.225} C_VEL
LIN {X 0,Y 573.697,Z 618.803,A -85,B 0,C 180,E1 -2045.122,E2 -2045.122} C_VEL
LIN {X 0,Y 573.526,Z 637.624,A -85,B 0,C 180,E1 -2048.091,E2 -2048.091} C_VEL
LIN {X 0,Y 573.493,Z 638.912,A -85,B 0,C 180,E1 -2048.292,E2 -2048.292} C_VEL
LIN {X 0,Y 574.583,Z 644.917,A -85,B 0,C 180,E1 -2048.405,E2 -2048.405} C_VEL
LIN {X 0,Y 574.253,Z 775.96,A -85,B 0,C 180,E1 -2050.086,E2 -2050.086} C_VEL
LIN {X 0,Y 574.159,Z 790.388,A -85,B 0,C 180,E1 -2050.422,E2 -2050.422} C_VEL
LIN {X 0,Y 574.028,Z 803.99,A -85,B 0,C 180,E1 -2050.882,E2 -2050.882} C_VEL
LIN {X 0,Y 573.812,Z 818.135,A -85,B 0,C 180,E1 -2051.524,E2 -2051.524} C_VEL
LIN {X 0,Y 573.702,Z 830.903,A -85,B 0,C 180,E1 -2052.268,E2 -2052.268} C_VEL
LIN {X 0,Y 573.537,Z 842.977,A -85,B 0,C 180,E1 -2053.137,E2 -2053.137} C_VEL
LIN {X 0,Y 573.421,Z 852.773,A -85,B 0,C 180,E1 -2053.992,E2 -2053.992} C_VEL
LIN {X 0,Y 573.271,Z 863.175,A -85,B 0,C 180,E1 -2055.081,E2 -2055.081} C_VEL
LIN {X 0,Y 573.175,Z 871.74,A -85,B 0,C 180,E1 -2056.167,E2 -2056.167} C_VEL
LIN {X 0,Y 573.106,Z 879.888,A -85,B 0,C 180,E1 -2057.428,E2 -2057.428} C_VEL
LIN {X 0,Y 573.015,Z 886.414,A -85,B 0,C 180,E1 -2058.683,E2 -2058.683} C_VEL
LIN {X 0,Y 573.002,Z 890.921,A -85,B 0,C 180,E1 -2059.756,E2 -2059.756} C_VEL
LIN {X 0,Y 572.969,Z 894.444,A -85,B 0,C 180,E1 -2060.825,E2 -2060.825} C_VEL
LIN {X 0,Y 572.979,Z 897.86,A -85,B 0,C 180,E1 -2062.246,E2 -2062.246} C_VEL
LIN {X 0,Y 572.974,Z 899.858,A -85,B 0,C 180,E1 -2063.662,E2 -2063.662} C_VEL
LIN {X 0,Y 572.932,Z 900.498,A -85,B 0,C 180,E1 -2065.074,E2 -2065.074} C_VEL
LIN {X 0,Y 572.977,Z 899.795,A -85,B 0,C 180,E1 -2066.484,E2 -2066.484} C_VEL
LIN {X 0,Y 572.938,Z 897.763,A -85,B 0,C 180,E1 -2067.891,E2 -2067.891} C_VEL
LIN {X 0,Y 572.946,Z 894.348,A -85,B 0,C 180,E1 -2069.297,E2 -2069.297} C_VEL
LIN {X 0,Y 572.984,Z 889.461,A -85,B 0,C 180,E1 -2070.703,E2 -2070.703} C_VEL
LIN {X 0,Y 573.031,Z 882.956,A -85,B 0,C 180,E1 -2072.109,E2 -2072.109} C_VEL
LIN {X 0,Y 573.141,Z 875.736,A -85,B 0,C 180,E1 -2073.339,E2 -2073.339} C_VEL
LIN {X 0,Y 573.255,Z 866.831,A -85,B 0,C 180,E1 -2074.571,E2 -2074.571} C_VEL
LIN {X 0,Y 573.354,Z 857.514,A -85,B 0,C 180,E1 -2075.628,E2 -2075.628} C_VEL
LIN {X 0,Y 573.523,Z 846.062,A -85,B 0,C 180,E1 -2076.696,E2 -2076.696} C_VEL
LIN {X 0,Y 573.679,Z 834.675,A -85,B 0,C 180,E1 -2077.568,E2 -2077.568} C_VEL
LIN {X 0,Y 573.841,Z 821.908,A -85,B 0,C 180,E1 -2078.363,E2 -2078.363} C_VEL
LIN {X 0,Y 574.003,Z 809.437,A -85,B 0,C 180,E1 -2078.981,E2 -2078.981} C_VEL
LIN {X 0,Y 574.142,Z 795.553,A -85,B 0,C 180,E1 -2079.512,E2 -2079.512} C_VEL
LIN {X 0,Y 574.225,Z 781.782,A -85,B 0,C 180,E1 -2079.889,E2 -2079.889} C_VEL
LIN {X 0,Y 574.257,Z 767.531,A -85,B 0,C 180,E1 -2080.133,E2 -2080.133} C_VEL
LIN {X 0,Y 574.57,Z 644.605,A -85,B 0,C 180,E1 -2081.689,E2 -2081.689} C_VEL
LIN {X 0,Y 573.501,Z 638.856,A -85,B 0,C 180,E1 -2081.807,E2 -2081.807} C_VEL
LIN {X 0,Y 573.664,Z 621.311,A -85,B 0,C 180,E1 -2084.57,E2 -2084.57} C_VEL
LIN {X 0,Y 573.664,Z 615.768,A -85,B 0,C 180,E1 -2085.454,E2 -2085.454} C_VEL
LIN {X 0,Y 573.222,Z 613.209,A -85,B 0,C 180,E1 -2085.899,E2 -2085.899} C_VEL
LIN {X 0,Y 573.195,Z 613.215,A -85,B 0,C 180,E1 -2088.59,E2 -2088.59} C_VEL
LIN {X 0,Y 573.255,Z 613.199,A -85,B 0,C 180,E1 -2091.29,E2 -2091.29} C_VEL
LIN {X 0,Y 573.198,Z 613.205,A -85,B 0,C 180,E1 -2093.867,E2 -2093.867} C_VEL
LIN {X 0,Y 573.194,Z 613.211,A -85,B 0,C 180,E1 -2096.483,E2 -2096.483} C_VEL
LIN {X 0,Y 573.229,Z 613.202,A -85,B 0,C 180,E1 -2099.368,E2 -2099.368} C_VEL
LIN {X 0,Y 573.233,Z 613.201,A -85,B 0,C 180,E1 -2102.224,E2 -2102.224} C_VEL
LIN {X 0,Y 573.188,Z 613.21,A -85,B 0,C 180,E1 -2105.189,E2 -2105.189} C_VEL
LIN {X 0,Y 573.218,Z 613.201,A -85,B 0,C 180,E1 -2107.809,E2 -2107.809} C_VEL
LIN {X 0,Y 573.214,Z 613.203,A -85,B 0,C 180,E1 -2110.528,E2 -2110.528} C_VEL
LIN {X 0,Y 573.203,Z 613.207,A -85,B 0,C 180,E1 -2113.363,E2 -2113.363} C_VEL
LIN {X 0,Y 573.207,Z 613.203,A -85,B 0,C 180,E1 -2116.335,E2 -2116.335} C_VEL
LIN {X 0,Y 573.249,Z 613.202,A -85,B 0,C 180,E1 -2119.475,E2 -2119.475} C_VEL
LIN {X 0,Y 573.217,Z 613.198,A -85,B 0,C 180,E1 -2122.191,E2 -2122.191} C_VEL
LIN {X 0,Y 573.229,Z 613.21,A -85,B 0,C 180,E1 -2125.23,E2 -2125.23} C_VEL
LIN {X 0,Y 573.238,Z 613.198,A -85,B 0,C 180,E1 -2128.184,E2 -2128.184} C_VEL
LIN {X 0,Y 573.241,Z 613.198,A -85,B 0,C 180,E1 -2130.632,E2 -2130.632} C_VEL
LIN {X 0,Y 573.204,Z 613.21,A -85,B 0,C 180,E1 -2133.515,E2 -2133.515} C_VEL
LIN {X 0,Y 573.218,Z 613.2,A -85,B 0,C 180,E1 -2136.134,E2 -2136.134} C_VEL
LIN {X 0,Y 573.253,Z 613.203,A -85,B 0,C 180,E1 -2139.173,E2 -2139.173} C_VEL
LIN {X 0,Y 573.22,Z 613.21,A -85,B 0,C 180,E1 -2141.411,E2 -2141.411} C_VEL
LIN {X 0,Y 573.244,Z 613.206,A -85,B 0,C 180,E1 -2143.621,E2 -2143.621} C_VEL
LIN {X 0,Y 573.275,Z 613.2,A -85,B 0,C 180,E1 -2145.807,E2 -2145.807} C_VEL
LIN {X 0,Y 573.267,Z 613.194,A -85,B 0,C 180,E1 -2148.745,E2 -2148.745} C_VEL
LIN {X 0,Y 573.282,Z 613.201,A -85,B 0,C 180,E1 -2151.54,E2 -2151.54} C_VEL
LIN {X 0,Y 573.282,Z 613.194,A -85,B 0,C 180,E1 -2154.372,E2 -2154.372} C_VEL
LIN {X 0,Y 573.313,Z 613.198,A -85,B 0,C 180,E1 -2157.892,E2 -2157.892} C_VEL
LIN {X 0,Y 573.332,Z 613.186,A -85,B 0,C 180,E1 -2160.702,E2 -2160.702} C_VEL
LIN {X 0,Y 573.307,Z 613.19,A -85,B 0,C 180,E1 -2162.81,E2 -2162.81} C_VEL
LIN {X 0,Y 573.287,Z 613.198,A -85,B 0,C 180,E1 -2165.628,E2 -2165.628} C_VEL
LIN {X 0,Y 573.286,Z 613.195,A -85,B 0,C 180,E1 -2168.459,E2 -2168.459} C_VEL
LIN {X 0,Y 573.275,Z 613.194,A -85,B 0,C 180,E1 -2171.312,E2 -2171.312} C_VEL
LIN {X 0,Y 573.285,Z 613.196,A -85,B 0,C 180,E1 -2174.424,E2 -2174.424} C_VEL
LIN {X 0,Y 573.262,Z 613.195,A -85,B 0,C 180,E1 -2177.111,E2 -2177.111} C_VEL
LIN {X 0,Y 573.256,Z 613.206,A -85,B 0,C 180,E1 -2180.076,E2 -2180.076} C_VEL
LIN {X 0,Y 573.238,Z 613.198,A -85,B 0,C 180,E1 -2183.099,E2 -2183.099} C_VEL
LIN {X 0,Y 573.255,Z 613.197,A -85,B 0,C 180,E1 -2185.41,E2 -2185.41} C_VEL
LIN {X 0,Y 573.255,Z 613.202,A -85,B 0,C 180,E1 -2188.029,E2 -2188.029} C_VEL
LIN {X 0,Y 573.236,Z 613.201,A -85,B 0,C 180,E1 -2190.883,E2 -2190.883} C_VEL
LIN {X 0,Y 573.265,Z 613.195,A -85,B 0,C 180,E1 -2193.524,E2 -2193.524} C_VEL
LIN {X 0,Y 573.219,Z 613.206,A -85,B 0,C 180,E1 -2196.051,E2 -2196.051} C_VEL
LIN {X 0,Y 573.251,Z 613.203,A -85,B 0,C 180,E1 -2198.701,E2 -2198.701} C_VEL
LIN {X 0,Y 573.238,Z 613.199,A -85,B 0,C 180,E1 -2201.456,E2 -2201.456} C_VEL
LIN {X 0,Y 573.238,Z 613.206,A -85,B 0,C 180,E1 -2204.333,E2 -2204.333} C_VEL
LIN {X 0,Y 573.243,Z 613.198,A -85,B 0,C 180,E1 -2207.358,E2 -2207.358} C_VEL
LIN {X 0,Y 573.243,Z 613.205,A -85,B 0,C 180,E1 -2210.392,E2 -2210.392} C_VEL
LIN {X 0,Y 573.258,Z 613.201,A -85,B 0,C 180,E1 -2213.078,E2 -2213.078} C_VEL
LIN {X 0,Y 573.276,Z 613.195,A -85,B 0,C 180,E1 -2215.672,E2 -2215.672} C_VEL
LIN {X 0,Y 573.251,Z 613.2,A -85,B 0,C 180,E1 -2218.185,E2 -2218.185} C_VEL
LIN {X 0,Y 573.268,Z 613.204,A -85,B 0,C 180,E1 -2220.634,E2 -2220.634} C_VEL
LIN {X 0,Y 573.273,Z 613.199,A -85,B 0,C 180,E1 -2223.501,E2 -2223.501} C_VEL
LIN {X 0,Y 573.308,Z 613.328,A -85,B 0,C 180,E1 -2225.006,E2 -2225.006} C_VEL
LIN {X 0,Y 574.399,Z 618.914,A -85,B 0,C 180,E1 -2225.802,E2 -2225.802} C_VEL
LIN {X 0,Y 574.06,Z 640.45,A -85,B 0,C 180,E1 -2228.623,E2 -2228.623} C_VEL
LIN {X 0,Y 573.839,Z 660.81,A -85,B 0,C 180,E1 -2231.247,E2 -2231.247} C_VEL
LIN {X 0,Y 573.666,Z 676.431,A -85,B 0,C 180,E1 -2233.233,E2 -2233.233} C_VEL
LIN {X 0,Y 574.594,Z 682.394,A -85,B 0,C 180,E1 -2233.341,E2 -2233.341} C_VEL
LIN {X 0,Y 574.271,Z 814.879,A -85,B 0,C 180,E1 -2235.04,E2 -2235.04} C_VEL
LIN {X 0,Y 574.145,Z 829.46,A -85,B 0,C 180,E1 -2235.379,E2 -2235.379} C_VEL
LIN {X 0,Y 573.996,Z 843.836,A -85,B 0,C 180,E1 -2235.87,E2 -2235.87} C_VEL
LIN {X 0,Y 573.871,Z 856.638,A -85,B 0,C 180,E1 -2236.454,E2 -2236.454} C_VEL
LIN {X 0,Y 573.719,Z 869.096,A -85,B 0,C 180,E1 -2237.172,E2 -2237.172} C_VEL
LIN {X 0,Y 573.566,Z 880.476,A -85,B 0,C 180,E1 -2237.977,E2 -2237.977} C_VEL
LIN {X 0,Y 573.449,Z 891.847,A -85,B 0,C 180,E1 -2238.955,E2 -2238.955} C_VEL
LIN {X 0,Y 573.268,Z 901.333,A -85,B 0,C 180,E1 -2239.939,E2 -2239.939} C_VEL
LIN {X 0,Y 573.197,Z 909.912,A -85,B 0,C 180,E1 -2241.006,E2 -2241.006} C_VEL
LIN {X 0,Y 573.111,Z 918.115,A -85,B 0,C 180,E1 -2242.248,E2 -2242.248} C_VEL
LIN {X 0,Y 573.035,Z 924.449,A -85,B 0,C 180,E1 -2243.427,E2 -2243.427} C_VEL
LIN {X 0,Y 573,Z 929.961,A -85,B 0,C 180,E1 -2244.722,E2 -2244.722} C_VEL
LIN {X 0,Y 573.029,Z 933.442,A -85,B 0,C 180,E1 -2245.78,E2 -2245.78} C_VEL
LIN {X 0,Y 572.956,Z 936.831,A -85,B 0,C 180,E1 -2247.188,E2 -2247.188} C_VEL
LIN {X 0,Y 572.941,Z 938.832,A -85,B 0,C 180,E1 -2248.594,E2 -2248.594} C_VEL
LIN {X 0,Y 572.936,Z 939.5,A -85,B 0,C 180,E1 -2250,E2 -2250} C_VEL
LIN {X 0,Y 572.941,Z 938.833,A -85,B 0,C 180,E1 -2251.406,E2 -2251.406} C_VEL
LIN {X 0,Y 572.956,Z 936.833,A -85,B 0,C 180,E1 -2252.812,E2 -2252.812} C_VEL
LIN {X 0,Y 573.029,Z 933.444,A -85,B 0,C 180,E1 -2254.22,E2 -2254.22} C_VEL
LIN {X 0,Y 573.059,Z 928.568,A -85,B 0,C 180,E1 -2255.63,E2 -2255.63} C_VEL
LIN {X 0,Y 573.058,Z 923.852,A -85,B 0,C 180,E1 -2256.693,E2 -2256.693} C_VEL
LIN {X 0,Y 573.126,Z 917.038,A -85,B 0,C 180,E1 -2257.929,E2 -2257.929} C_VEL
LIN {X 0,Y 573.225,Z 908.559,A -85,B 0,C 180,E1 -2259.171,E2 -2259.171} C_VEL
LIN {X 0,Y 573.304,Z 899.708,A -85,B 0,C 180,E1 -2260.239,E2 -2260.239} C_VEL
LIN {X 0,Y 573.462,Z 888.992,A -85,B 0,C 180,E1 -2261.308,E2 -2261.308} C_VEL
LIN {X 0,Y 573.612,Z 878.145,A -85,B 0,C 180,E1 -2262.201,E2 -2262.201} C_VEL
LIN {X 0,Y 573.76,Z 866.261,A -85,B 0,C 180,E1 -2263.007,E2 -2263.007} C_VEL
LIN {X 0,Y 573.939,Z 853.095,A -85,B 0,C 180,E1 -2263.724,E2 -2263.724} C_VEL
LIN {X 0,Y 574.076,Z 839.831,A -85,B 0,C 180,E1 -2264.284,E2 -2264.284} C_VEL
LIN {X 0,Y 574.2,Z 825.832,A -85,B 0,C 180,E1 -2264.72,E2 -2264.72} C_VEL
LIN {X 0,Y 574.303,Z 812.133,A -85,B 0,C 180,E1 -2265.005,E2 -2265.005} C_VEL
LIN {X 0,Y 574.531,Z 681.288,A -85,B 0,C 180,E1 -2266.675,E2 -2266.675} C_VEL
LIN {X 0,Y 573.648,Z 676.342,A -85,B 0,C 180,E1 -2266.779,E2 -2266.779} C_VEL
LIN {X 0,Y 573.869,Z 655.466,A -85,B 0,C 180,E1 -2269.439,E2 -2269.439} C_VEL
LIN {X 0,Y 574.145,Z 634.807,A -85,B 0,C 180,E1 -2272.111,E2 -2272.111} C_VEL
LIN {X 0,Y 574.398,Z 618.915,A -85,B 0,C 180,E1 -2274.198,E2 -2274.198} C_VEL
LIN {X 0,Y 573.285,Z 613.201,A -85,B 0,C 180,E1 -2275.032,E2 -2275.032} C_VEL
LIN {X 0,Y 573.291,Z 613.196,A -85,B 0,C 180,E1 -2277.765,E2 -2277.765} C_VEL
LIN {X 0,Y 573.252,Z 613.198,A -85,B 0,C 180,E1 -2280.176,E2 -2280.176} C_VEL
LIN {X 0,Y 573.258,Z 613.198,A -85,B 0,C 180,E1 -2282.645,E2 -2282.645} C_VEL
LIN {X 0,Y 573.271,Z 613.203,A -85,B 0,C 180,E1 -2285.183,E2 -2285.183} C_VEL
LIN {X 0,Y 573.238,Z 613.202,A -85,B 0,C 180,E1 -2287.807,E2 -2287.807} C_VEL
